LIN {X 0,Y 600.05,Z 1006.774,A -85,B 0,C 180,E1 28192.716,E2 28192.716} C_VEL
LIN {X 0,Y 598.178,Z 1023.897,A -85,B 0,C 180,E1 28190.857,E2 28190.857} C_VEL
LIN {X 0,Y 596.63,Z 1038.34,A -85,B 0,C 180,E1 28189.054,E2 28189.054} C_VEL
LIN {X 0,Y 595.296,Z 1052.251,A -85,B 0,C 180,E1 28187.094,E2 28187.094} C_VEL
LIN {X 0,Y 594.084,Z 1066.083,A -85,B 0,C 180,E1 28184.823,E2 28184.823} C_VEL
LIN {X 0,Y 593.249,Z 1077.838,A -85,B 0,C 180,E1 28182.61,E2 28182.61} C_VEL
LIN {X 0,Y 592.685,Z 1087.23,A -85,B 0,C 180,E1 28180.498,E2 28180.498} C_VEL
LIN {X 0,Y 592.308,Z 1095.363,A -85,B 0,C 180,E1 28178.348,E2 28178.348} C_VEL
LIN {X 0,Y 592.058,Z 1102.422,A -85,B 0,C 180,E1 28176.01,E2 28176.01} C_VEL
LIN {X 0,Y 591.967,Z 1107.243,A -85,B 0,C 180,E1 28173.971,E2 28173.971} C_VEL
LIN {X 0,Y 591.915,Z 1111.392,A -85,B 0,C 180,E1 28171.549,E2 28171.549} C_VEL
LIN {X 0,Y 591.912,Z 1113.53,A -85,B 0,C 180,E1 28169.419,E2 28169.419} C_VEL
LIN {X 0,Y 591.896,Z 1114.429,A -85,B 0,C 180,E1 28167.289,E2 28167.289} C_VEL
LIN {X 0,Y 591.895,Z 1113.793,A -85,B 0,C 180,E1 28164.863,E2 28164.863} C_VEL
LIN {X 0,Y 591.889,Z 1112.043,A -85,B 0,C 180,E1 28162.916,E2 28162.916} C_VEL
LIN {X 0,Y 591.93,Z 1109.042,A -85,B 0,C 180,E1 28160.864,E2 28160.864} C_VEL
LIN {X 0,Y 592.028,Z 1103.73,A -85,B 0,C 180,E1 28158.402,E2 28158.402} C_VEL
LIN {X 0,Y 592.196,Z 1098.141,A -85,B 0,C 180,E1 28156.426,E2 28156.426} C_VEL
LIN {X 0,Y 592.531,Z 1090.169,A -85,B 0,C 180,E1 28154.128,E2 28154.128} C_VEL
LIN {X 0,Y 593.026,Z 1080.989,A -85,B 0,C 180,E1 28151.981,E2 28151.981} C_VEL
LIN {X 0,Y 593.774,Z 1070.166,A -85,B 0,C 180,E1 28149.805,E2 28149.805} C_VEL
LIN {X 0,Y 594.831,Z 1057.029,A -85,B 0,C 180,E1 28147.568,E2 28147.568} C_VEL
LIN {X 0,Y 596.239,Z 1042.636,A -85,B 0,C 180,E1 28145.424,E2 28145.424} C_VEL
LIN {X 0,Y 597.762,Z 1027.606,A -85,B 0,C 180,E1 28143.497,E2 28143.497} C_VEL
LIN {X 0,Y 599.626,Z 1011.06,A -85,B 0,C 180,E1 28141.625,E2 28141.625} C_VEL
LIN {X 0,Y 601.534,Z 993.698,A -85,B 0,C 180,E1 28139.927,E2 28139.927} C_VEL
LIN {X 0,Y 603.744,Z 974.807,A -85,B 0,C 180,E1 28138.298,E2 28138.298} C_VEL
LIN {X 0,Y 605.898,Z 955.015,A -85,B 0,C 180,E1 28136.834,E2 28136.834} C_VEL
LIN {X 0,Y 608.034,Z 935.172,A -85,B 0,C 180,E1 28135.549,E2 28135.549} C_VEL
LIN {X 0,Y 610.125,Z 913.844,A -85,B 0,C 180,E1 28134.377,E2 28134.377} C_VEL
LIN {X 0,Y 611.917,Z 894.087,A -85,B 0,C 180,E1 28133.444,E2 28133.444} C_VEL
LIN {X 0,Y 613.892,Z 869.658,A -85,B 0,C 180,E1 28132.487,E2 28132.487} C_VEL
LIN {X 0,Y 615.266,Z 849.158,A -85,B 0,C 180,E1 28131.836,E2 28131.836} C_VEL
LIN {X 0,Y 616.599,Z 825.684,A -85,B 0,C 180,E1 28131.244,E2 28131.244} C_VEL
LIN {X 0,Y 617.493,Z 801.735,A -85,B 0,C 180,E1 28130.817,E2 28130.817} C_VEL
LIN {X 0,Y 622.364,Z 560.753,A -85,B 0,C 180,E1 28127.651,E2 28127.651} C_VEL
LIN {X 0,Y 624.229,Z 467.095,A -85,B 0,C 180,E1 28126.398,E2 28126.398} C_VEL
LIN {X 0,Y 610.775,Z 444.903,A -85,B 0,C 180,E1 28124.91,E2 28124.91} C_VEL
LIN {X 0,Y 602.614,Z 432.977,A -85,B 0,C 180,E1 28123.98,E2 28123.98} C_VEL
LIN {X 0,Y 599.127,Z 428.129,A -85,B 0,C 180,E1 28123.572,E2 28123.572} C_VEL
LIN {X 0,Y 596.004,Z 423.491,A -85,B 0,C 180,E1 28123.195,E2 28123.195} C_VEL
LIN {X 0,Y 593.804,Z 420.57,A -85,B 0,C 180,E1 28122.932,E2 28122.932} C_VEL
LIN {X 0,Y 593.243,Z 418.839,A -85,B 0,C 180,E1 28122.785,E2 28122.785} C_VEL
LIN {X 0,Y 593.129,Z 418.323,A -85,B 0,C 180,E1 28122.532,E2 28122.532} C_VEL
LIN {X 0,Y 593.115,Z 418.332,A -85,B 0,C 180,E1 28119.712,E2 28119.712} C_VEL
LIN {X 0,Y 593.141,Z 418.28,A -85,B 0,C 180,E1 28116.518,E2 28116.518} C_VEL
LIN {X 0,Y 593.127,Z 418.344,A -85,B 0,C 180,E1 28113.569,E2 28113.569} C_VEL
LIN {X 0,Y 593.136,Z 418.28,A -85,B 0,C 180,E1 28110.268,E2 28110.268} C_VEL
LIN {X 0,Y 593.14,Z 418.328,A -85,B 0,C 180,E1 28107.401,E2 28107.401} C_VEL
LIN {X 0,Y 593.144,Z 418.327,A -85,B 0,C 180,E1 28104.076,E2 28104.076} C_VEL
LIN {X 0,Y 593.163,Z 418.336,A -85,B 0,C 180,E1 28101.146,E2 28101.146} C_VEL
LIN {X 0,Y 593.149,Z 418.343,A -85,B 0,C 180,E1 28097.867,E2 28097.867} C_VEL
LIN {X 0,Y 593.202,Z 418.328,A -85,B 0,C 180,E1 28094.745,E2 28094.745} C_VEL
LIN {X 0,Y 593.148,Z 418.326,A -85,B 0,C 180,E1 28091.572,E2 28091.572} C_VEL
LIN {X 0,Y 593.199,Z 418.334,A -85,B 0,C 180,E1 28088.433,E2 28088.433} C_VEL
LIN {X 0,Y 593.159,Z 418.335,A -85,B 0,C 180,E1 28085.32,E2 28085.32} C_VEL
LIN {X 0,Y 593.189,Z 418.315,A -85,B 0,C 180,E1 28082.029,E2 28082.029} C_VEL
LIN {X 0,Y 593.193,Z 418.332,A -85,B 0,C 180,E1 28078.744,E2 28078.744} C_VEL
LIN {X 0,Y 593.172,Z 418.334,A -85,B 0,C 180,E1 28075.456,E2 28075.456} C_VEL
LIN {X 0,Y 593.189,Z 418.32,A -85,B 0,C 180,E1 28072.25,E2 28072.25} C_VEL
LIN {X 0,Y 593.178,Z 418.335,A -85,B 0,C 180,E1 28069.019,E2 28069.019} C_VEL
LIN {X 0,Y 593.199,Z 418.336,A -85,B 0,C 180,E1 28065.747,E2 28065.747} C_VEL
LIN {X 0,Y 593.19,Z 418.327,A -85,B 0,C 180,E1 28062.439,E2 28062.439} C_VEL
LIN {X 0,Y 593.183,Z 418.32,A -85,B 0,C 180,E1 28059.165,E2 28059.165} C_VEL
LIN {X 0,Y 593.18,Z 418.342,A -85,B 0,C 180,E1 28056.011,E2 28056.011} C_VEL
LIN {X 0,Y 593.188,Z 418.313,A -85,B 0,C 180,E1 28052.819,E2 28052.819} C_VEL
LIN {X 0,Y 593.177,Z 418.329,A -85,B 0,C 180,E1 28049.622,E2 28049.622} C_VEL
LIN {X 0,Y 593.187,Z 418.342,A -85,B 0,C 180,E1 28046.319,E2 28046.319} C_VEL
LIN {X 0,Y 593.197,Z 418.338,A -85,B 0,C 180,E1 28043.033,E2 28043.033} C_VEL
LIN {X 0,Y 593.161,Z 418.331,A -85,B 0,C 180,E1 28039.914,E2 28039.914} C_VEL
LIN {X 0,Y 593.211,Z 418.506,A -85,B 0,C 180,E1 28037.12,E2 28037.12} C_VEL
LIN {X 0,Y 597.822,Z 429.519,A -85,B 0,C 180,E1 28035.508,E2 28035.508} C_VEL
LIN {X 0,Y 605.197,Z 447.603,A -85,B 0,C 180,E1 28033.091,E2 28033.091} C_VEL
LIN {X 0,Y 606.689,Z 450.565,A -85,B 0,C 180,E1 28032.827,E2 28032.827} C_VEL
LIN {X 0,Y 617.614,Z 468.823,A -85,B 0,C 180,E1 28031.586,E2 28031.586} C_VEL
LIN {X 0,Y 620.789,Z 474.786,A -85,B 0,C 180,E1 28031.228,E2 28031.228} C_VEL
LIN {X 0,Y 624.171,Z 491.358,A -85,B 0,C 180,E1 28030.702,E2 28030.702} C_VEL
LIN {X 0,Y 619.361,Z 729.252,A -85,B 0,C 180,E1 28027.569,E2 28027.569} C_VEL
LIN {X 0,Y 617.111,Z 841.64,A -85,B 0,C 180,E1 28026.088,E2 28026.088} C_VEL
LIN {X 0,Y 615.922,Z 867.301,A -85,B 0,C 180,E1 28025.592,E2 28025.592} C_VEL
LIN {X 0,Y 614.631,Z 888.381,A -85,B 0,C 180,E1 28025.045,E2 28025.045} C_VEL
LIN {X 0,Y 612.923,Z 912.524,A -85,B 0,C 180,E1 28024.251,E2 28024.251} C_VEL
LIN {X 0,Y 611.154,Z 933.412,A -85,B 0,C 180,E1 28023.404,E2 28023.404} C_VEL
LIN {X 0,Y 609.26,Z 954.504,A -85,B 0,C 180,E1 28022.401,E2 28022.401} C_VEL
LIN {X 0,Y 607.047,Z 976.733,A -85,B 0,C 180,E1 28021.145,E2 28021.145} C_VEL
LIN {X 0,Y 605.079,Z 996.004,A -85,B 0,C 180,E1 28019.888,E2 28019.888} C_VEL
LIN {X 0,Y 602.838,Z 1016.85,A -85,B 0,C 180,E1 28018.319,E2 28018.319} C_VEL
LIN {X 0,Y 601,Z 1033.899,A -85,B 0,C 180,E1 28016.853,E2 28016.853} C_VEL
LIN {X 0,Y 598.954,Z 1053.455,A -85,B 0,C 180,E1 28014.931,E2 28014.931} C_VEL
LIN {X 0,Y 597.428,Z 1068.492,A -85,B 0,C 180,E1 28013.242,E2 28013.242} C_VEL
LIN {X 0,Y 595.881,Z 1084.893,A -85,B 0,C 180,E1 28011.148,E2 28011.148} C_VEL
LIN {X 0,Y 594.747,Z 1097.865,A -85,B 0,C 180,E1 28009.239,E2 28009.239} C_VEL
LIN {X 0,Y 593.777,Z 1110.217,A -85,B 0,C 180,E1 28007.139,E2 28007.139} C_VEL
LIN {X 0,Y 593.037,Z 1121.053,A -85,B 0,C 180,E1 28004.959,E2 28004.959} C_VEL
LIN {X 0,Y 592.515,Z 1130.773,A -85,B 0,C 180,E1 28002.673,E2 28002.673} C_VEL
LIN {X 0,Y 592.187,Z 1138.512,A -85,B 0,C 180,E1 28000.409,E2 28000.409} C_VEL
LIN {X 0,Y 592.024,Z 1144.591,A -85,B 0,C 180,E1 27998.222,E2 27998.222} C_VEL
LIN {X 0,Y 591.937,Z 1149.494,A -85,B 0,C 180,E1 27995.817,E2 27995.817} C_VEL
LIN {X 0,Y 591.915,Z 1152.349,A -85,B 0,C 180,E1 27993.777,E2 27993.777} C_VEL
LIN {X 0,Y 591.903,Z 1154.19,A -85,B 0,C 180,E1 27991.355,E2 27991.355} C_VEL
LIN {X 0,Y 591.885,Z 1154.349,A -85,B 0,C 180,E1 27989.322,E2 27989.322} C_VEL
LIN {X 0,Y 591.888,Z 1153.358,A -85,B 0,C 180,E1 27987.289,E2 27987.289} C_VEL
LIN {X 0,Y 591.902,Z 1150.611,A -85,B 0,C 180,E1 27984.863,E2 27984.863} C_VEL
LIN {X 0,Y 591.969,Z 1146.895,A -85,B 0,C 180,E1 27982.82,E2 27982.82} C_VEL
LIN {X 0,Y 592.092,Z 1141.711,A -85,B 0,C 180,E1 27980.67,E2 27980.67} C_VEL
LIN {X 0,Y 592.34,Z 1134.306,A -85,B 0,C 180,E1 27978.313,E2 27978.313} C_VEL
LIN {X 0,Y 592.697,Z 1126.746,A -85,B 0,C 180,E1 27976.339,E2 27976.339} C_VEL
LIN {X 0,Y 593.332,Z 1116.399,A -85,B 0,C 180,E1 27974.056,E2 27974.056} C_VEL
LIN {X 0,Y 594.113,Z 1105.682,A -85,B 0,C 180,E1 27972.062,E2 27972.062} C_VEL
LIN {X 0,Y 595.076,Z 1093.997,A -85,B 0,C 180,E1 27970.159,E2 27970.159} C_VEL
LIN {X 0,Y 596.424,Z 1078.851,A -85,B 0,C 180,E1 27968.046,E2 27968.046} C_VEL
LIN {X 0,Y 597.795,Z 1064.893,A -85,B 0,C 180,E1 27966.332,E2 27966.332} C_VEL
LIN {X 0,Y 599.722,Z 1046.098,A -85,B 0,C 180,E1 27964.311,E2 27964.311} C_VEL
LIN {X 0,Y 601.503,Z 1029.441,A -85,B 0,C 180,E1 27962.744,E2 27962.744} C_VEL
LIN {X 0,Y 603.743,Z 1008.537,A -85,B 0,C 180,E1 27961.025,E2 27961.025} C_VEL
LIN {X 0,Y 605.691,Z 989.997,A -85,B 0,C 180,E1 27959.699,E2 27959.699} C_VEL
LIN {X 0,Y 608.024,Z 967.457,A -85,B 0,C 180,E1 27958.304,E2 27958.304} C_VEL
LIN {X 0,Y 609.822,Z 948.512,A -85,B 0,C 180,E1 27957.298,E2 27957.298} C_VEL
LIN {X 0,Y 611.747,Z 927.152,A -85,B 0,C 180,E1 27956.32,E2 27956.32} C_VEL
LIN {X 0,Y 613.509,Z 903.939,A -85,B 0,C 180,E1 27955.447,E2 27955.447} C_VEL
LIN {X 0,Y 614.991,Z 882.112,A -85,B 0,C 180,E1 27954.779,E2 27954.779} C_VEL
LIN {X 0,Y 616.42,Z 856.718,A -85,B 0,C 180,E1 27954.191,E2 27954.191} C_VEL
LIN {X 0,Y 617.238,Z 834.898,A -85,B 0,C 180,E1 27953.824,E2 27953.824} C_VEL
LIN {X 0,Y 621.554,Z 599.011,A -85,B 0,C 180,E1 27950.762,E2 27950.762} C_VEL
LIN {X 0,Y 623.531,Z 489.86,A -85,B 0,C 180,E1 27949.324,E2 27949.324} C_VEL
LIN {X 0,Y 619.644,Z 473.187,A -85,B 0,C 180,E1 27948.779,E2 27948.779} C_VEL
LIN {X 0,Y 605.414,Z 448.968,A -85,B 0,C 180,E1 27947.25,E2 27947.25} C_VEL
LIN {X 0,Y 597.591,Z 429.213,A -85,B 0,C 180,E1 27944.783,E2 27944.783} C_VEL
LIN {X 0,Y 593.228,Z 418.535,A -85,B 0,C 180,E1 27943.318,E2 27943.318} C_VEL
LIN {X 0,Y 593.154,Z 418.284,A -85,B 0,C 180,E1 27940.34,E2 27940.34} C_VEL
LIN {X 0,Y 593.193,Z 418.324,A -85,B 0,C 180,E1 27937.239,E2 27937.239} C_VEL
LIN {X 0,Y 593.167,Z 418.338,A -85,B 0,C 180,E1 27934.031,E2 27934.031} C_VEL
LIN {X 0,Y 593.202,Z 418.338,A -85,B 0,C 180,E1 27930.723,E2 27930.723} C_VEL
LIN {X 0,Y 593.195,Z 418.331,A -85,B 0,C 180,E1 27927.398,E2 27927.398} C_VEL
LIN {X 0,Y 593.177,Z 418.316,A -85,B 0,C 180,E1 27924.181,E2 27924.181} C_VEL
LIN {X 0,Y 593.185,Z 418.337,A -85,B 0,C 180,E1 27921.041,E2 27921.041} C_VEL
LIN {X 0,Y 593.183,Z 418.33,A -85,B 0,C 180,E1 27917.764,E2 27917.764} C_VEL
LIN {X 0,Y 593.184,Z 418.318,A -85,B 0,C 180,E1 27914.546,E2 27914.546} C_VEL
LIN {X 0,Y 593.187,Z 418.341,A -85,B 0,C 180,E1 27911.175,E2 27911.175} C_VEL
LIN {X 0,Y 593.191,Z 418.317,A -85,B 0,C 180,E1 27907.945,E2 27907.945} C_VEL
LIN {X 0,Y 593.169,Z 418.332,A -85,B 0,C 180,E1 27904.738,E2 27904.738} C_VEL
LIN {X 0,Y 593.193,Z 418.329,A -85,B 0,C 180,E1 27901.545,E2 27901.545} C_VEL
LIN {X 0,Y 593.167,Z 418.325,A -85,B 0,C 180,E1 27898.409,E2 27898.409} C_VEL
LIN {X 0,Y 593.182,Z 418.343,A -85,B 0,C 180,E1 27895.068,E2 27895.068} C_VEL
LIN {X 0,Y 593.189,Z 418.313,A -85,B 0,C 180,E1 27891.86,E2 27891.86} C_VEL
LIN {X 0,Y 593.155,Z 418.34,A -85,B 0,C 180,E1 27888.625,E2 27888.625} C_VEL
LIN {X 0,Y 593.2,Z 418.317,A -85,B 0,C 180,E1 27885.454,E2 27885.454} C_VEL
LIN {X 0,Y 593.144,Z 418.334,A -85,B 0,C 180,E1 27882.336,E2 27882.336} C_VEL
LIN {X 0,Y 593.199,Z 418.335,A -85,B 0,C 180,E1 27879.166,E2 27879.166} C_VEL
LIN {X 0,Y 593.136,Z 418.318,A -85,B 0,C 180,E1 27876.135,E2 27876.135} C_VEL
LIN {X 0,Y 593.177,Z 418.335,A -85,B 0,C 180,E1 27872.927,E2 27872.927} C_VEL
LIN {X 0,Y 593.132,Z 418.342,A -85,B 0,C 180,E1 27869.955,E2 27869.955} C_VEL
LIN {X 0,Y 593.156,Z 418.328,A -85,B 0,C 180,E1 27866.732,E2 27866.732} C_VEL
LIN {X 0,Y 593.125,Z 418.338,A -85,B 0,C 180,E1 27863.841,E2 27863.841} C_VEL
LIN {X 0,Y 593.152,Z 418.339,A -85,B 0,C 180,E1 27860.666,E2 27860.666} C_VEL
LIN {X 0,Y 593.104,Z 418.276,A -85,B 0,C 180,E1 27857.858,E2 27857.858} C_VEL
LIN {X 0,Y 593.152,Z 418.346,A -85,B 0,C 180,E1 27854.653,E2 27854.653} C_VEL
LIN {X 0,Y 593.097,Z 418.282,A -85,B 0,C 180,E1 27851.682,E2 27851.682} C_VEL
LIN {X 0,Y 593.209,Z 418.548,A -85,B 0,C 180,E1 27850.844,E2 27850.844} C_VEL
LIN {X 0,Y 593.536,Z 419.937,A -85,B 0,C 180,E1 27850.687,E2 27850.687} C_VEL
LIN {X 0,Y 595.547,Z 423.115,A -85,B 0,C 180,E1 27850.449,E2 27850.449} C_VEL
LIN {X 0,Y 596.796,Z 424.91,A -85,B 0,C 180,E1 27850.31,E2 27850.31} C_VEL
LIN {X 0,Y 607.889,Z 441.301,A -85,B 0,C 180,E1 27849.107,E2 27849.107} C_VEL
LIN {X 0,Y 623.849,Z 467.241,A -85,B 0,C 180,E1 27847.442,E2 27847.442} C_VEL
LIN {X 0,Y 622.311,Z 544.948,A -85,B 0,C 180,E1 27846.423,E2 27846.423} C_VEL
LIN {X 0,Y 621.357,Z 552.646,A -85,B 0,C 180,E1 27846.382,E2 27846.382} C_VEL
LIN {X 0,Y 616.074,Z 573.201,A -85,B 0,C 180,E1 27846.476,E2 27846.476} C_VEL
LIN {X 0,Y 615.373,Z 579.803,A -85,B 0,C 180,E1 27846.432,E2 27846.432} C_VEL
LIN {X 0,Y 610.821,Z 804.731,A -85,B 0,C 180,E1 27843.476,E2 27843.476} C_VEL
LIN {X 0,Y 609.717,Z 830.998,A -85,B 0,C 180,E1 27842.97,E2 27842.97} C_VEL
LIN {X 0,Y 608.493,Z 851.442,A -85,B 0,C 180,E1 27842.436,E2 27842.436} C_VEL
LIN {X 0,Y 606.891,Z 874.614,A -85,B 0,C 180,E1 27841.679,E2 27841.679} C_VEL
LIN {X 0,Y 604.931,Z 896.78,A -85,B 0,C 180,E1 27840.774,E2 27840.774} C_VEL
LIN {X 0,Y 602.985,Z 917.369,A -85,B 0,C 180,E1 27839.778,E2 27839.778} C_VEL
LIN {X 0,Y 600.686,Z 938.996,A -85,B 0,C 180,E1 27838.538,E2 27838.538} C_VEL
LIN {X 0,Y 598.657,Z 957.009,A -85,B 0,C 180,E1 27837.343,E2 27837.343} C_VEL
LIN {X 0,Y 596.2,Z 977.938,A -85,B 0,C 180,E1 27835.745,E2 27835.745} C_VEL
LIN {X 0,Y 594.122,Z 994.981,A -85,B 0,C 180,E1 27834.245,E2 27834.245} C_VEL
LIN {X 0,Y 592.002,Z 1013.013,A -85,B 0,C 180,E1 27832.44,E2 27832.44} C_VEL
LIN {X 0,Y 590.145,Z 1028.649,A -85,B 0,C 180,E1 27830.635,E2 27830.635} C_VEL
LIN {X 0,Y 588.491,Z 1043.984,A -85,B 0,C 180,E1 27828.628,E2 27828.628} C_VEL
LIN {X 0,Y 587.102,Z 1057.157,A -85,B 0,C 180,E1 27826.626,E2 27826.626} C_VEL
LIN {X 0,Y 586.026,Z 1069.289,A -85,B 0,C 180,E1 27824.526,E2 27824.526} C_VEL
LIN {X 0,Y 585.142,Z 1080.722,A -85,B 0,C 180,E1 27822.194,E2 27822.194} C_VEL
LIN {X 0,Y 584.612,Z 1089.812,A -85,B 0,C 180,E1 27820.047,E2 27820.047} C_VEL
LIN {X 0,Y 584.237,Z 1098.008,A -85,B 0,C 180,E1 27817.672,E2 27817.672} C_VEL
LIN {X 0,Y 584.035,Z 1103.796,A -85,B 0,C 180,E1 27815.6,E2 27815.6} C_VEL
LIN {X 0,Y 583.929,Z 1109.024,A -85,B 0,C 180,E1 27813.141,E2 27813.141} C_VEL
LIN {X 0,Y 583.893,Z 1112.005,A -85,B 0,C 180,E1 27811.079,E2 27811.079} C_VEL
LIN {X 0,Y 583.9,Z 1113.762,A -85,B 0,C 180,E1 27809.117,E2 27809.117} C_VEL
LIN {X 0,Y 583.895,Z 1114.44,A -85,B 0,C 180,E1 27806.662,E2 27806.662} C_VEL
LIN {X 0,Y 583.908,Z 1113.559,A -85,B 0,C 180,E1 27804.497,E2 27804.497} C_VEL
LIN {X 0,Y 583.925,Z 1111.424,A -85,B 0,C 180,E1 27802.324,E2 27802.324} C_VEL
LIN {X 0,Y 583.977,Z 1107.242,A -85,B 0,C 180,E1 27799.842,E2 27799.842} C_VEL
LIN {X 0,Y 584.067,Z 1102.564,A -85,B 0,C 180,E1 27797.83,E2 27797.83} C_VEL
LIN {X 0,Y 584.339,Z 1095.46,A -85,B 0,C 180,E1 27795.431,E2 27795.431} C_VEL
LIN {X 0,Y 584.754,Z 1087.143,A -85,B 0,C 180,E1 27793.203,E2 27793.203} C_VEL
LIN {X 0,Y 585.402,Z 1077.256,A -85,B 0,C 180,E1 27790.959,E2 27790.959} C_VEL
LIN {X 0,Y 586.294,Z 1066.066,A -85,B 0,C 180,E1 27788.804,E2 27788.804} C_VEL
LIN {X 0,Y 587.469,Z 1053.823,A -85,B 0,C 180,E1 27786.742,E2 27786.742} C_VEL
LIN {X 0,Y 588.944,Z 1039.5,A -85,B 0,C 180,E1 27784.669,E2 27784.669} C_VEL
LIN {X 0,Y 590.513,Z 1025.638,A -85,B 0,C 180,E1 27782.904,E2 27782.904} C_VEL
LIN {X 0,Y 592.594,Z 1007.842,A -85,B 0,C 180,E1 27780.925,E2 27780.925} C_VEL
LIN {X 0,Y 594.618,Z 991.223,A -85,B 0,C 180,E1 27779.312,E2 27779.312} C_VEL
LIN {X 0,Y 597.05,Z 970.874,A -85,B 0,C 180,E1 27777.594,E2 27777.594} C_VEL
LIN {X 0,Y 599.106,Z 953.171,A -85,B 0,C 180,E1 27776.294,E2 27776.294} C_VEL
LIN {X 0,Y 601.587,Z 931.163,A -85,B 0,C 180,E1 27774.894,E2 27774.894} C_VEL
LIN {X 0,Y 603.541,Z 912.109,A -85,B 0,C 180,E1 27773.858,E2 27773.858} C_VEL
LIN {X 0,Y 605.588,Z 890.917,A -85,B 0,C 180,E1 27772.864,E2 27772.864} C_VEL
LIN {X 0,Y 607.464,Z 867.705,A -85,B 0,C 180,E1 27771.974,E2 27771.974} C_VEL
LIN {X 0,Y 608.969,Z 846.238,A -85,B 0,C 180,E1 27771.301,E2 27771.301} C_VEL
LIN {X 0,Y 610.364,Z 821.032,A -85,B 0,C 180,E1 27770.701,E2 27770.701} C_VEL
LIN {X 0,Y 611.203,Z 799.034,A -85,B 0,C 180,E1 27770.323,E2 27770.323} C_VEL
LIN {X 0,Y 616.602,Z 546.316,A -85,B 0,C 180,E1 27766.975,E2 27766.975} C_VEL
LIN {X 0,Y 618.221,Z 470.366,A -85,B 0,C 180,E1 27765.949,E2 27765.949} C_VEL
LIN {X 0,Y 605.233,Z 449.14,A -85,B 0,C 180,E1 27764.482,E2 27764.482} C_VEL
LIN {X 0,Y 597.704,Z 438.133,A -85,B 0,C 180,E1 27763.603,E2 27763.603} C_VEL
LIN {X 0,Y 591.444,Z 429.254,A -85,B 0,C 180,E1 27762.847,E2 27762.847} C_VEL
LIN {X 0,Y 588.36,Z 424.737,A -85,B 0,C 180,E1 27762.463,E2 27762.463} C_VEL
LIN {X 0,Y 585.933,Z 421.842,A -85,B 0,C 180,E1 27762.167,E2 27762.167} C_VEL
LIN {X 0,Y 585.242,Z 419.789,A -85,B 0,C 180,E1 27761.995,E2 27761.995} C_VEL
LIN {X 0,Y 585.172,Z 419.275,A -85,B 0,C 180,E1 27761.659,E2 27761.659} C_VEL
LIN {X 0,Y 585.186,Z 419.32,A -85,B 0,C 180,E1 27758.334,E2 27758.334} C_VEL
LIN {X 0,Y 585.194,Z 419.272,A -85,B 0,C 180,E1 27755.397,E2 27755.397} C_VEL
LIN {X 0,Y 585.19,Z 419.323,A -85,B 0,C 180,E1 27752.1,E2 27752.1} C_VEL
LIN {X 0,Y 585.22,Z 419.262,A -85,B 0,C 180,E1 27749.14,E2 27749.14} C_VEL
LIN {X 0,Y 585.197,Z 419.335,A -85,B 0,C 180,E1 27745.939,E2 27745.939} C_VEL
LIN {X 0,Y 585.26,Z 419.323,A -85,B 0,C 180,E1 27742.819,E2 27742.819} C_VEL
LIN {X 0,Y 585.201,Z 419.317,A -85,B 0,C 180,E1 27739.67,E2 27739.67} C_VEL
LIN {X 0,Y 585.258,Z 419.308,A -85,B 0,C 180,E1 27736.476,E2 27736.476} C_VEL
LIN {X 0,Y 585.215,Z 419.334,A -85,B 0,C 180,E1 27733.336,E2 27733.336} C_VEL
LIN {X 0,Y 585.237,Z 419.327,A -85,B 0,C 180,E1 27730.036,E2 27730.036} C_VEL
LIN {X 0,Y 585.247,Z 419.31,A -85,B 0,C 180,E1 27726.869,E2 27726.869} C_VEL
LIN {X 0,Y 585.225,Z 419.328,A -85,B 0,C 180,E1 27723.624,E2 27723.624} C_VEL
LIN {X 0,Y 585.257,Z 419.323,A -85,B 0,C 180,E1 27720.392,E2 27720.392} C_VEL
LIN {X 0,Y 585.227,Z 419.307,A -85,B 0,C 180,E1 27717.16,E2 27717.16} C_VEL
LIN {X 0,Y 585.255,Z 419.317,A -85,B 0,C 180,E1 27713.821,E2 27713.821} C_VEL
LIN {X 0,Y 585.254,Z 419.33,A -85,B 0,C 180,E1 27710.461,E2 27710.461} C_VEL
LIN {X 0,Y 585.236,Z 419.31,A -85,B 0,C 180,E1 27707.167,E2 27707.167} C_VEL
LIN {X 0,Y 585.245,Z 419.314,A -85,B 0,C 180,E1 27704.034,E2 27704.034} C_VEL
LIN {X 0,Y 585.252,Z 419.332,A -85,B 0,C 180,E1 27700.747,E2 27700.747} C_VEL
LIN {X 0,Y 585.258,Z 419.306,A -85,B 0,C 180,E1 27697.393,E2 27697.393} C_VEL
LIN {X 0,Y 585.239,Z 419.309,A -85,B 0,C 180,E1 27694.172,E2 27694.172} C_VEL
LIN {X 0,Y 585.252,Z 419.329,A -85,B 0,C 180,E1 27690.974,E2 27690.974} C_VEL
LIN {X 0,Y 585.23,Z 419.314,A -85,B 0,C 180,E1 27687.787,E2 27687.787} C_VEL
LIN {X 0,Y 585.255,Z 419.306,A -85,B 0,C 180,E1 27684.582,E2 27684.582} C_VEL
LIN {X 0,Y 585.241,Z 419.311,A -85,B 0,C 180,E1 27681.333,E2 27681.333} C_VEL
LIN {X 0,Y 585.23,Z 419.357,A -85,B 0,C 180,E1 27678.006,E2 27678.006} C_VEL
LIN {X 0,Y 585.303,Z 419.848,A -85,B 0,C 180,E1 27677.785,E2 27677.785} C_VEL
LIN {X 0,Y 592.102,Z 435.669,A -85,B 0,C 180,E1 27675.45,E2 27675.45} C_VEL
LIN {X 0,Y 597.515,Z 448.594,A -85,B 0,C 180,E1 27673.719,E2 27673.719} C_VEL
LIN {X 0,Y 610.489,Z 470.096,A -85,B 0,C 180,E1 27672.179,E2 27672.179} C_VEL
LIN {X 0,Y 615.277,Z 478.799,A -85,B 0,C 180,E1 27671.63,E2 27671.63} C_VEL
LIN {X 0,Y 618.124,Z 493.199,A -85,B 0,C 180,E1 27671.168,E2 27671.168} C_VEL
LIN {X 0,Y 613.047,Z 730.309,A -85,B 0,C 180,E1 27668.017,E2 27668.017} C_VEL
LIN {X 0,Y 610.688,Z 841.32,A -85,B 0,C 180,E1 27666.539,E2 27666.539} C_VEL
LIN {X 0,Y 609.414,Z 867.194,A -85,B 0,C 180,E1 27666.036,E2 27666.036} C_VEL
LIN {X 0,Y 608.038,Z 888.463,A -85,B 0,C 180,E1 27665.478,E2 27665.478} C_VEL
LIN {X 0,Y 606.24,Z 912.394,A -85,B 0,C 180,E1 27664.682,E2 27664.682} C_VEL
LIN {X 0,Y 604.378,Z 933.221,A -85,B 0,C 180,E1 27663.829,E2 27663.829} C_VEL
LIN {X 0,Y 602.37,Z 954.246,A -85,B 0,C 180,E1 27662.818,E2 27662.818} C_VEL
LIN {X 0,Y 600.014,Z 976.431,A -85,B 0,C 180,E1 27661.552,E2 27661.552} C_VEL
LIN {X 0,Y 597.92,Z 995.771,A -85,B 0,C 180,E1 27660.278,E2 27660.278} C_VEL
LIN {X 0,Y 595.564,Z 1016.545,A -85,B 0,C 180,E1 27658.696,E2 27658.696} C_VEL
LIN {X 0,Y 593.589,Z 1033.748,A -85,B 0,C 180,E1 27657.201,E2 27657.201} C_VEL
LIN {X 0,Y 591.377,Z 1053.62,A -85,B 0,C 180,E1 27655.219,E2 27655.219} C_VEL
LIN {X 0,Y 589.732,Z 1068.861,A -85,B 0,C 180,E1 27653.481,E2 27653.481} C_VEL
LIN {X 0,Y 588.039,Z 1085.699,A -85,B 0,C 180,E1 27651.281,E2 27651.281} C_VEL
LIN {X 0,Y 586.881,Z 1098.212,A -85,B 0,C 180,E1 27649.404,E2 27649.404} C_VEL
LIN {X 0,Y 585.79,Z 1111.701,A -85,B 0,C 180,E1 27647.073,E2 27647.073} C_VEL
LIN {X 0,Y 585.131,Z 1121.094,A -85,B 0,C 180,E1 27645.156,E2 27645.156} C_VEL
LIN {X 0,Y 584.57,Z 1130.783,A -85,B 0,C 180,E1 27642.845,E2 27642.845} C_VEL
LIN {X 0,Y 584.217,Z 1138.512,A -85,B 0,C 180,E1 27640.552,E2 27640.552} C_VEL
LIN {X 0,Y 584.036,Z 1144.718,A -85,B 0,C 180,E1 27638.286,E2 27638.286} C_VEL
LIN {X 0,Y 583.944,Z 1149.494,A -85,B 0,C 180,E1 27635.897,E2 27635.897} C_VEL
LIN {X 0,Y 583.915,Z 1152.349,A -85,B 0,C 180,E1 27633.829,E2 27633.829} C_VEL
LIN {X 0,Y 583.902,Z 1154.19,A -85,B 0,C 180,E1 27631.374,E2 27631.374} C_VEL
LIN {X 0,Y 583.885,Z 1154.348,A -85,B 0,C 180,E1 27629.313,E2 27629.313} C_VEL
LIN {X 0,Y 583.89,Z 1153.426,A -85,B 0,C 180,E1 27627.35,E2 27627.35} C_VEL
LIN {X 0,Y 583.905,Z 1150.929,A -85,B 0,C 180,E1 27624.99,E2 27624.99} C_VEL
LIN {X 0,Y 583.971,Z 1147.101,A -85,B 0,C 180,E1 27622.82,E2 27622.82} C_VEL
LIN {X 0,Y 584.086,Z 1142.219,A -85,B 0,C 180,E1 27620.74,E2 27620.74} C_VEL
LIN {X 0,Y 584.365,Z 1134.658,A -85,B 0,C 180,E1 27618.251,E2 27618.251} C_VEL
LIN {X 0,Y 584.746,Z 1127.072,A -85,B 0,C 180,E1 27616.23,E2 27616.23} C_VEL
LIN {X 0,Y 585.417,Z 1116.912,A -85,B 0,C 180,E1 27613.937,E2 27613.937} C_VEL
LIN {X 0,Y 586.225,Z 1106.102,A -85,B 0,C 180,E1 27611.915,E2 27611.915} C_VEL
LIN {X 0,Y 587.232,Z 1094.351,A -85,B 0,C 180,E1 27609.986,E2 27609.986} C_VEL
LIN {X 0,Y 588.656,Z 1079.34,A -85,B 0,C 180,E1 27607.846,E2 27607.846} C_VEL
LIN {X 0,Y 590.1,Z 1065.458,A -85,B 0,C 180,E1 27606.11,E2 27606.11} C_VEL
LIN {X 0,Y 592.031,Z 1047.857,A -85,B 0,C 180,E1 27604.167,E2 27604.167} C_VEL
LIN {X 0,Y 593.957,Z 1030.723,A -85,B 0,C 180,E1 27602.521,E2 27602.521} C_VEL
LIN {X 0,Y 596.169,Z 1011.618,A -85,B 0,C 180,E1 27600.897,E2 27600.897} C_VEL
LIN {X 0,Y 598.313,Z 992.123,A -85,B 0,C 180,E1 27599.467,E2 27599.467} C_VEL
LIN {X 0,Y 600.595,Z 971.593,A -85,B 0,C 180,E1 27598.146,E2 27598.146} C_VEL
LIN {X 0,Y 602.753,Z 950.216,A -85,B 0,C 180,E1 27596.979,E2 27596.979} C_VEL
LIN {X 0,Y 604.474,Z 931.982,A -85,B 0,C 180,E1 27596.12,E2 27596.12} C_VEL
LIN {X 0,Y 606.477,Z 908.711,A -85,B 0,C 180,E1 27595.19,E2 27595.19} C_VEL
LIN {X 0,Y 608.102,Z 885.734,A -85,B 0,C 180,E1 27594.457,E2 27594.457} C_VEL
LIN {X 0,Y 609.617,Z 861.627,A -85,B 0,C 180,E1 27593.853,E2 27593.853} C_VEL
LIN {X 0,Y 610.635,Z 837.267,A -85,B 0,C 180,E1 27593.424,E2 27593.424} C_VEL
LIN {X 0,Y 615.209,Z 602.161,A -85,B 0,C 180,E1 27590.342,E2 27590.342} C_VEL
LIN {X 0,Y 617.3,Z 491.496,A -85,B 0,C 180,E1 27588.868,E2 27588.868} C_VEL
LIN {X 0,Y 613.962,Z 477.24,A -85,B 0,C 180,E1 27588.394,E2 27588.394} C_VEL
LIN {X 0,Y 599.58,Z 452.97,A -85,B 0,C 180,E1 27586.835,E2 27586.835} C_VEL
LIN {X 0,Y 596.897,Z 448.207,A -85,B 0,C 180,E1 27586.489,E2 27586.489} C_VEL
LIN {X 0,Y 589.654,Z 430.249,A -85,B 0,C 180,E1 27584.168,E2 27584.168} C_VEL
LIN {X 0,Y 585.256,Z 419.491,A -85,B 0,C 180,E1 27582.651,E2 27582.651} C_VEL
LIN {X 0,Y 585.241,Z 419.287,A -85,B 0,C 180,E1 27579.716,E2 27579.716} C_VEL
LIN {X 0,Y 585.23,Z 419.312,A -85,B 0,C 180,E1 27576.416,E2 27576.416} C_VEL
LIN {X 0,Y 585.255,Z 419.31,A -85,B 0,C 180,E1 27573.259,E2 27573.259} C_VEL
LIN {X 0,Y 585.229,Z 419.327,A -85,B 0,C 180,E1 27570.04,E2 27570.04} C_VEL
LIN {X 0,Y 585.255,Z 419.328,A -85,B 0,C 180,E1 27566.81,E2 27566.81} C_VEL
LIN {X 0,Y 585.255,Z 419.306,A -85,B 0,C 180,E1 27563.443,E2 27563.443} C_VEL
LIN {X 0,Y 585.247,Z 419.32,A -85,B 0,C 180,E1 27560.189,E2 27560.189} C_VEL
LIN {X 0,Y 585.244,Z 419.33,A -85,B 0,C 180,E1 27556.909,E2 27556.909} C_VEL
LIN {X 0,Y 585.244,Z 419.304,A -85,B 0,C 180,E1 27553.738,E2 27553.738} C_VEL
LIN {X 0,Y 585.243,Z 419.323,A -85,B 0,C 180,E1 27550.534,E2 27550.534} C_VEL
LIN {X 0,Y 585.249,Z 419.319,A -85,B 0,C 180,E1 27547.165,E2 27547.165} C_VEL
LIN {X 0,Y 585.253,Z 419.31,A -85,B 0,C 180,E1 27543.919,E2 27543.919} C_VEL
LIN {X 0,Y 585.227,Z 419.331,A -85,B 0,C 180,E1 27540.685,E2 27540.685} C_VEL
LIN {X 0,Y 585.253,Z 419.303,A -85,B 0,C 180,E1 27537.454,E2 27537.454} C_VEL
LIN {X 0,Y 585.229,Z 419.328,A -85,B 0,C 180,E1 27534.214,E2 27534.214} C_VEL
LIN {X 0,Y 585.227,Z 419.314,A -85,B 0,C 180,E1 27530.857,E2 27530.857} C_VEL
LIN {X 0,Y 585.256,Z 419.319,A -85,B 0,C 180,E1 27527.669,E2 27527.669} C_VEL
LIN {X 0,Y 585.21,Z 419.332,A -85,B 0,C 180,E1 27524.505,E2 27524.505} C_VEL
LIN {X 0,Y 585.259,Z 419.306,A -85,B 0,C 180,E1 27521.368,E2 27521.368} C_VEL
LIN {X 0,Y 585.2,Z 419.331,A -85,B 0,C 180,E1 27518.237,E2 27518.237} C_VEL
LIN {X 0,Y 585.247,Z 419.312,A -85,B 0,C 180,E1 27515.039,E2 27515.039} C_VEL
LIN {X 0,Y 585.196,Z 419.318,A -85,B 0,C 180,E1 27511.974,E2 27511.974} C_VEL
LIN {X 0,Y 585.214,Z 419.33,A -85,B 0,C 180,E1 27508.682,E2 27508.682} C_VEL
LIN {X 0,Y 585.201,Z 419.331,A -85,B 0,C 180,E1 27505.677,E2 27505.677} C_VEL
LIN {X 0,Y 585.19,Z 419.326,A -85,B 0,C 180,E1 27502.411,E2 27502.411} C_VEL
LIN {X 0,Y 585.184,Z 419.295,A -85,B 0,C 180,E1 27499.64,E2 27499.64} C_VEL
LIN {X 0,Y 585.173,Z 419.287,A -85,B 0,C 180,E1 27496.285,E2 27496.285} C_VEL
LIN {X 0,Y 585.186,Z 419.289,A -85,B 0,C 180,E1 27493.384,E2 27493.384} C_VEL
LIN {X 0,Y 585.189,Z 419.452,A -85,B 0,C 180,E1 27491.585,E2 27491.585} C_VEL
LIN {X 0,Y 585.536,Z 420.845,A -85,B 0,C 180,E1 27491.402,E2 27491.402} C_VEL
LIN {X 0,Y 587.43,Z 423.887,A -85,B 0,C 180,E1 27491.168,E2 27491.168} C_VEL
LIN {X 0,Y 588.76,Z 425.467,A -85,B 0,C 180,E1 27491.021,E2 27491.021} C_VEL
LIN {X 0,Y 591.543,Z 429.527,A -85,B 0,C 180,E1 27490.702,E2 27490.702} C_VEL
LIN {X 0,Y 605.321,Z 450.203,A -85,B 0,C 180,E1 27489.183,E2 27489.183} C_VEL
LIN {X 0,Y 617.641,Z 470.603,A -85,B 0,C 180,E1 27487.874,E2 27487.874} C_VEL
LIN {X 0,Y 615.373,Z 579.803,A -85,B 0,C 180,E1 27486.432,E2 27486.432} C_VEL
LIN {X 0,Y 614.451,Z 587.499,A -85,B 0,C 180,E1 27486.388,E2 27486.388} C_VEL
LIN {X 0,Y 609.124,Z 608.05,A -85,B 0,C 180,E1 27486.486,E2 27486.486} C_VEL
LIN {X 0,Y 608.406,Z 614.655,A -85,B 0,C 180,E1 27486.442,E2 27486.442} C_VEL
LIN {X 0,Y 604.328,Z 805.826,A -85,B 0,C 180,E1 27483.907,E2 27483.907} C_VEL
LIN {X 0,Y 603.172,Z 831.725,A -85,B 0,C 180,E1 27483.399,E2 27483.399} C_VEL
LIN {X 0,Y 601.898,Z 852.117,A -85,B 0,C 180,E1 27482.861,E2 27482.861} C_VEL
LIN {X 0,Y 600.227,Z 875.132,A -85,B 0,C 180,E1 27482.101,E2 27482.101} C_VEL
LIN {X 0,Y 598.234,Z 896.836,A -85,B 0,C 180,E1 27481.207,E2 27481.207} C_VEL
LIN {X 0,Y 596.306,Z 916.322,A -85,B 0,C 180,E1 27480.263,E2 27480.263} C_VEL
LIN {X 0,Y 593.783,Z 939.121,A -85,B 0,C 180,E1 27478.956,E2 27478.956} C_VEL
LIN {X 0,Y 591.567,Z 957.896,A -85,B 0,C 180,E1 27477.698,E2 27477.698} C_VEL
LIN {X 0,Y 588.906,Z 979.323,A -85,B 0,C 180,E1 27476.034,E2 27476.034} C_VEL
LIN {X 0,Y 586.799,Z 995.731,A -85,B 0,C 180,E1 27474.568,E2 27474.568} C_VEL
LIN {X 0,Y 584.554,Z 1013.69,A -85,B 0,C 180,E1 27472.742,E2 27472.742} C_VEL
LIN {X 0,Y 582.596,Z 1029.29,A -85,B 0,C 180,E1 27470.915,E2 27470.915} C_VEL
LIN {X 0,Y 580.831,Z 1044.568,A -85,B 0,C 180,E1 27468.883,E2 27468.883} C_VEL
LIN {X 0,Y 579.357,Z 1057.713,A -85,B 0,C 180,E1 27466.855,E2 27466.855} C_VEL
LIN {X 0,Y 578.211,Z 1069.817,A -85,B 0,C 180,E1 27464.727,E2 27464.727} C_VEL
LIN {X 0,Y 577.303,Z 1080.504,A -85,B 0,C 180,E1 27462.504,E2 27462.504} C_VEL
LIN {X 0,Y 576.718,Z 1089.234,A -85,B 0,C 180,E1 27460.388,E2 27460.388} C_VEL
LIN {X 0,Y 576.283,Z 1097.535,A -85,B 0,C 180,E1 27457.979,E2 27457.979} C_VEL
LIN {X 0,Y 576.056,Z 1103.398,A -85,B 0,C 180,E1 27455.878,E2 27455.878} C_VEL
LIN {X 0,Y 575.94,Z 1108.444,A -85,B 0,C 180,E1 27453.583,E2 27453.583} C_VEL
LIN {X 0,Y 575.9,Z 1111.827,A -85,B 0,C 180,E1 27451.293,E2 27451.293} C_VEL
LIN {X 0,Y 575.91,Z 1113.655,A -85,B 0,C 180,E1 27449.304,E2 27449.304} C_VEL
LIN {X 0,Y 575.904,Z 1114.497,A -85,B 0,C 180,E1 27446.915,E2 27446.915} C_VEL
LIN {X 0,Y 575.907,Z 1113.666,A -85,B 0,C 180,E1 27444.62,E2 27444.62} C_VEL
LIN {X 0,Y 575.899,Z 1111.831,A -85,B 0,C 180,E1 27442.618,E2 27442.618} C_VEL
LIN {X 0,Y 575.942,Z 1108.402,A -85,B 0,C 180,E1 27440.305,E2 27440.305} C_VEL
LIN {X 0,Y 576.049,Z 1103.519,A -85,B 0,C 180,E1 27438.079,E2 27438.079} C_VEL
LIN {X 0,Y 576.268,Z 1097.876,A -85,B 0,C 180,E1 27436.044,E2 27436.044} C_VEL
LIN {X 0,Y 576.701,Z 1089.478,A -85,B 0,C 180,E1 27433.584,E2 27433.584} C_VEL
LIN {X 0,Y 577.3,Z 1080.554,A -85,B 0,C 180,E1 27431.416,E2 27431.416} C_VEL
LIN {X 0,Y 578.239,Z 1069.547,A -85,B 0,C 180,E1 27429.132,E2 27429.132} C_VEL
LIN {X 0,Y 579.369,Z 1057.658,A -85,B 0,C 180,E1 27427.043,E2 27427.043} C_VEL
LIN {X 0,Y 580.903,Z 1044.07,A -85,B 0,C 180,E1 27424.948,E2 27424.948} C_VEL
LIN {X 0,Y 582.648,Z 1028.964,A -85,B 0,C 180,E1 27422.95,E2 27422.95} C_VEL
LIN {X 0,Y 584.611,Z 1013.384,A -85,B 0,C 180,E1 27421.129,E2 27421.129} C_VEL
LIN {X 0,Y 586.845,Z 995.508,A -85,B 0,C 180,E1 27419.316,E2 27419.316} C_VEL
LIN {X 0,Y 589.056,Z 978.397,A -85,B 0,C 180,E1 27417.792,E2 27417.792} C_VEL
LIN {X 0,Y 591.667,Z 957.309,A -85,B 0,C 180,E1 27416.162,E2 27416.162} C_VEL
LIN {X 0,Y 593.914,Z 938.555,A -85,B 0,C 180,E1 27414.906,E2 27414.906} C_VEL
LIN {X 0,Y 596.471,Z 915.739,A -85,B 0,C 180,E1 27413.599,E2 27413.599} C_VEL
LIN {X 0,Y 598.426,Z 896.448,A -85,B 0,C 180,E1 27412.661,E2 27412.661} C_VEL
LIN {X 0,Y 600.54,Z 873.751,A -85,B 0,C 180,E1 27411.729,E2 27411.729} C_VEL
LIN {X 0,Y 602.205,Z 851.292,A -85,B 0,C 180,E1 27410.99,E2 27410.99} C_VEL
LIN {X 0,Y 603.559,Z 830.091,A -85,B 0,C 180,E1 27410.432,E2 27410.432} C_VEL
LIN {X 0,Y 604.689,Z 804.624,A -85,B 0,C 180,E1 27409.943,E2 27409.943} C_VEL
LIN {X 0,Y 610.012,Z 570.914,A -85,B 0,C 180,E1 27406.81,E2 27406.81} C_VEL
LIN {X 0,Y 612.177,Z 473.5,A -85,B 0,C 180,E1 27405.483,E2 27405.483} C_VEL
LIN {X 0,Y 599.275,Z 452.543,A -85,B 0,C 180,E1 27403.989,E2 27403.989} C_VEL
LIN {X 0,Y 590.483,Z 439.918,A -85,B 0,C 180,E1 27402.934,E2 27402.934} C_VEL
LIN {X 0,Y 583.996,Z 430.758,A -85,B 0,C 180,E1 27402.124,E2 27402.124} C_VEL
LIN {X 0,Y 581.244,Z 426.926,A -85,B 0,C 180,E1 27401.773,E2 27401.773} C_VEL
LIN {X 0,Y 580.331,Z 425.644,A -85,B 0,C 180,E1 27401.655,E2 27401.655} C_VEL
LIN {X 0,Y 578.027,Z 422.821,A -85,B 0,C 180,E1 27401.361,E2 27401.361} C_VEL
LIN {X 0,Y 577.368,Z 420.81,A -85,B 0,C 180,E1 27401.189,E2 27401.189} C_VEL
LIN {X 0,Y 577.299,Z 420.266,A -85,B 0,C 180,E1 27400.897,E2 27400.897} C_VEL
LIN {X 0,Y 577.232,Z 420.29,A -85,B 0,C 180,E1 27397.948,E2 27397.948} C_VEL
LIN {X 0,Y 577.302,Z 420.266,A -85,B 0,C 180,E1 27394.817,E2 27394.817} C_VEL
LIN {X 0,Y 577.243,Z 420.294,A -85,B 0,C 180,E1 27391.733,E2 27391.733} C_VEL
LIN {X 0,Y 577.297,Z 420.256,A -85,B 0,C 180,E1 27388.557,E2 27388.557} C_VEL
LIN {X 0,Y 577.26,Z 420.325,A -85,B 0,C 180,E1 27385.519,E2 27385.519} C_VEL
LIN {X 0,Y 577.281,Z 420.321,A -85,B 0,C 180,E1 27382.185,E2 27382.185} C_VEL
LIN {X 0,Y 577.289,Z 420.308,A -85,B 0,C 180,E1 27379.109,E2 27379.109} C_VEL
LIN {X 0,Y 577.272,Z 420.298,A -85,B 0,C 180,E1 27375.883,E2 27375.883} C_VEL
LIN {X 0,Y 577.314,Z 420.31,A -85,B 0,C 180,E1 27372.809,E2 27372.809} C_VEL
LIN {X 0,Y 577.275,Z 420.319,A -85,B 0,C 180,E1 27369.572,E2 27369.572} C_VEL
LIN {X 0,Y 577.321,Z 420.297,A -85,B 0,C 180,E1 27366.364,E2 27366.364} C_VEL
LIN {X 0,Y 577.288,Z 420.311,A -85,B 0,C 180,E1 27363.177,E2 27363.177} C_VEL
LIN {X 0,Y 577.304,Z 420.313,A -85,B 0,C 180,E1 27359.802,E2 27359.802} C_VEL
LIN {X 0,Y 577.314,Z 420.297,A -85,B 0,C 180,E1 27356.525,E2 27356.525} C_VEL
LIN {X 0,Y 577.291,Z 420.303,A -85,B 0,C 180,E1 27353.236,E2 27353.236} C_VEL
LIN {X 0,Y 577.315,Z 420.315,A -85,B 0,C 180,E1 27350.026,E2 27350.026} C_VEL
LIN {X 0,Y 577.315,Z 420.303,A -85,B 0,C 180,E1 27346.682,E2 27346.682} C_VEL
LIN {X 0,Y 577.308,Z 420.297,A -85,B 0,C 180,E1 27343.395,E2 27343.395} C_VEL
LIN {X 0,Y 577.303,Z 420.311,A -85,B 0,C 180,E1 27340.133,E2 27340.133} C_VEL
LIN {X 0,Y 577.31,Z 420.304,A -85,B 0,C 180,E1 27336.849,E2 27336.849} C_VEL
LIN {X 0,Y 577.309,Z 420.288,A -85,B 0,C 180,E1 27333.565,E2 27333.565} C_VEL
LIN {X 0,Y 577.301,Z 420.313,A -85,B 0,C 180,E1 27330.192,E2 27330.192} C_VEL
LIN {X 0,Y 577.318,Z 420.315,A -85,B 0,C 180,E1 27326.936,E2 27326.936} C_VEL
LIN {X 0,Y 577.29,Z 420.304,A -85,B 0,C 180,E1 27323.649,E2 27323.649} C_VEL
LIN {X 0,Y 577.315,Z 420.295,A -85,B 0,C 180,E1 27320.404,E2 27320.404} C_VEL
LIN {X 0,Y 577.365,Z 420.606,A -85,B 0,C 180,E1 27318.581,E2 27318.581} C_VEL
LIN {X 0,Y 584.328,Z 436.973,A -85,B 0,C 180,E1 27316.088,E2 27316.088} C_VEL
LIN {X 0,Y 588.858,Z 447.813,A -85,B 0,C 180,E1 27314.576,E2 27314.576} C_VEL
LIN {X 0,Y 600.324,Z 466.222,A -85,B 0,C 180,E1 27313.153,E2 27313.153} C_VEL
LIN {X 0,Y 609.83,Z 482.982,A -85,B 0,C 180,E1 27312.034,E2 27312.034} C_VEL
LIN {X 0,Y 612.136,Z 494.978,A -85,B 0,C 180,E1 27311.647,E2 27311.647} C_VEL
LIN {X 0,Y 606.782,Z 731.117,A -85,B 0,C 180,E1 27308.479,E2 27308.479} C_VEL
LIN {X 0,Y 604.312,Z 841.013,A -85,B 0,C 180,E1 27307.001,E2 27307.001} C_VEL
LIN {X 0,Y 602.967,Z 866.903,A -85,B 0,C 180,E1 27306.495,E2 27306.495} C_VEL
LIN {X 0,Y 601.503,Z 888.401,A -85,B 0,C 180,E1 27305.927,E2 27305.927} C_VEL
LIN {X 0,Y 599.6,Z 912.332,A -85,B 0,C 180,E1 27305.122,E2 27305.122} C_VEL
LIN {X 0,Y 597.637,Z 933.188,A -85,B 0,C 180,E1 27304.259,E2 27304.259} C_VEL
LIN {X 0,Y 595.534,Z 953.982,A -85,B 0,C 180,E1 27303.249,E2 27303.249} C_VEL
LIN {X 0,Y 593.03,Z 976.197,A -85,B 0,C 180,E1 27301.967,E2 27301.967} C_VEL
LIN {X 0,Y 590.808,Z 995.409,A -85,B 0,C 180,E1 27300.687,E2 27300.687} C_VEL
LIN {X 0,Y 588.315,Z 1016.239,A -85,B 0,C 180,E1 27299.083,E2 27299.083} C_VEL
LIN {X 0,Y 586.246,Z 1033.289,A -85,B 0,C 180,E1 27297.585,E2 27297.585} C_VEL
LIN {X 0,Y 583.93,Z 1052.847,A -85,B 0,C 180,E1 27295.618,E2 27295.618} C_VEL
LIN {X 0,Y 582.216,Z 1067.7,A -85,B 0,C 180,E1 27293.91,E2 27293.91} C_VEL
LIN {X 0,Y 580.485,Z 1083.814,A -85,B 0,C 180,E1 27291.808,E2 27291.808} C_VEL
LIN {X 0,Y 579.191,Z 1096.62,A -85,B 0,C 180,E1 27289.883,E2 27289.883} C_VEL
LIN {X 0,Y 578.104,Z 1109.29,A -85,B 0,C 180,E1 27287.723,E2 27287.723} C_VEL
LIN {X 0,Y 577.249,Z 1120.445,A -85,B 0,C 180,E1 27285.471,E2 27285.471} C_VEL
LIN {X 0,Y 576.684,Z 1129.564,A -85,B 0,C 180,E1 27283.333,E2 27283.333} C_VEL
LIN {X 0,Y 576.264,Z 1137.906,A -85,B 0,C 180,E1 27280.902,E2 27280.902} C_VEL
LIN {X 0,Y 576.054,Z 1143.491,A -85,B 0,C 180,E1 27278.887,E2 27278.887} C_VEL
LIN {X 0,Y 575.953,Z 1148.695,A -85,B 0,C 180,E1 27276.479,E2 27276.479} C_VEL
LIN {X 0,Y 575.922,Z 1152.007,A -85,B 0,C 180,E1 27274.182,E2 27274.182} C_VEL
LIN {X 0,Y 575.91,Z 1153.902,A -85,B 0,C 180,E1 27271.99,E2 27271.99} C_VEL
LIN {X 0,Y 575.885,Z 1154.393,A -85,B 0,C 180,E1 27269.503,E2 27269.503} C_VEL
LIN {X 0,Y 575.893,Z 1153.493,A -85,B 0,C 180,E1 27267.413,E2 27267.413} C_VEL
LIN {X 0,Y 575.91,Z 1151.211,A -85,B 0,C 180,E1 27265.12,E2 27265.12} C_VEL
LIN {X 0,Y 575.974,Z 1147.308,A -85,B 0,C 180,E1 27262.82,E2 27262.82} C_VEL
LIN {X 0,Y 576.082,Z 1142.728,A -85,B 0,C 180,E1 27260.812,E2 27260.812} C_VEL
LIN {X 0,Y 576.336,Z 1136.069,A -85,B 0,C 180,E1 27258.491,E2 27258.491} C_VEL
LIN {X 0,Y 576.739,Z 1128.325,A -85,B 0,C 180,E1 27256.362,E2 27256.362} C_VEL
LIN {X 0,Y 577.311,Z 1119.518,A -85,B 0,C 180,E1 27254.324,E2 27254.324} C_VEL
LIN {X 0,Y 578.283,Z 1106.977,A -85,B 0,C 180,E1 27251.866,E2 27251.866} C_VEL
LIN {X 0,Y 579.324,Z 1095.35,A -85,B 0,C 180,E1 27249.912,E2 27249.912} C_VEL
LIN {X 0,Y 580.817,Z 1080.611,A -85,B 0,C 180,E1 27247.745,E2 27247.745} C_VEL
LIN {X 0,Y 582.414,Z 1066.022,A -85,B 0,C 180,E1 27245.883,E2 27245.883} C_VEL
LIN {X 0,Y 584.343,Z 1049.604,A -85,B 0,C 180,E1 27244.02,E2 27244.02} C_VEL
LIN {X 0,Y 586.509,Z 1031.305,A -85,B 0,C 180,E1 27242.227,E2 27242.227} C_VEL
LIN {X 0,Y 588.824,Z 1012.411,A -85,B 0,C 180,E1 27240.591,E2 27240.591} C_VEL
LIN {X 0,Y 591.137,Z 992.563,A -85,B 0,C 180,E1 27239.112,E2 27239.112} C_VEL
LIN {X 0,Y 593.425,Z 972.888,A -85,B 0,C 180,E1 27237.829,E2 27237.829} C_VEL
LIN {X 0,Y 595.792,Z 950.825,A -85,B 0,C 180,E1 27236.601,E2 27236.601} C_VEL
LIN {X 0,Y 597.704,Z 931.529,A -85,B 0,C 180,E1 27235.683,E2 27235.683} C_VEL
LIN {X 0,Y 599.794,Z 908.171,A -85,B 0,C 180,E1 27234.745,E2 27234.745} C_VEL
LIN {X 0,Y 601.497,Z 885.325,A -85,B 0,C 180,E1 27234.013,E2 27234.013} C_VEL
LIN {X 0,Y 603.097,Z 861.01,A -85,B 0,C 180,E1 27233.403,E2 27233.403} C_VEL
LIN {X 0,Y 604.146,Z 836.827,A -85,B 0,C 180,E1 27232.976,E2 27232.976} C_VEL
LIN {X 0,Y 608.969,Z 601.524,A -85,B 0,C 180,E1 27229.863,E2 27229.863} C_VEL
LIN {X 0,Y 611.131,Z 493.266,A -85,B 0,C 180,E1 27228.411,E2 27228.411} C_VEL
LIN {X 0,Y 608.335,Z 481.313,A -85,B 0,C 180,E1 27228.005,E2 27228.005} C_VEL
LIN {X 0,Y 591.765,Z 453.323,A -85,B 0,C 180,E1 27226.159,E2 27226.159} C_VEL
LIN {X 0,Y 588.684,Z 448.253,A -85,B 0,C 180,E1 27225.789,E2 27225.789} C_VEL
LIN {X 0,Y 581.508,Z 430.723,A -85,B 0,C 180,E1 27223.456,E2 27223.456} C_VEL
LIN {X 0,Y 577.31,Z 420.467,A -85,B 0,C 180,E1 27221.964,E2 27221.964} C_VEL
LIN {X 0,Y 577.319,Z 420.301,A -85,B 0,C 180,E1 27219.082,E2 27219.082} C_VEL
LIN {X 0,Y 577.295,Z 420.307,A -85,B 0,C 180,E1 27215.833,E2 27215.833} C_VEL
LIN {X 0,Y 577.301,Z 420.3,A -85,B 0,C 180,E1 27212.475,E2 27212.475} C_VEL
LIN {X 0,Y 577.314,Z 420.295,A -85,B 0,C 180,E1 27209.237,E2 27209.237} C_VEL
LIN {X 0,Y 577.3,Z 420.321,A -85,B 0,C 180,E1 27205.984,E2 27205.984} C_VEL
LIN {X 0,Y 577.314,Z 420.309,A -85,B 0,C 180,E1 27202.72,E2 27202.72} C_VEL
LIN {X 0,Y 577.313,Z 420.295,A -85,B 0,C 180,E1 27199.423,E2 27199.423} C_VEL
LIN {X 0,Y 577.311,Z 420.316,A -85,B 0,C 180,E1 27196.088,E2 27196.088} C_VEL
LIN {X 0,Y 577.301,Z 420.305,A -85,B 0,C 180,E1 27192.911,E2 27192.911} C_VEL
LIN {X 0,Y 577.309,Z 420.3,A -85,B 0,C 180,E1 27189.672,E2 27189.672} C_VEL
LIN {X 0,Y 577.306,Z 420.315,A -85,B 0,C 180,E1 27186.364,E2 27186.364} C_VEL
LIN {X 0,Y 577.296,Z 420.293,A -85,B 0,C 180,E1 27182.978,E2 27182.978} C_VEL
LIN {X 0,Y 577.319,Z 420.318,A -85,B 0,C 180,E1 27179.702,E2 27179.702} C_VEL
LIN {X 0,Y 577.285,Z 420.306,A -85,B 0,C 180,E1 27176.425,E2 27176.425} C_VEL
LIN {X 0,Y 577.312,Z 420.301,A -85,B 0,C 180,E1 27173.136,E2 27173.136} C_VEL
LIN {X 0,Y 577.31,Z 420.312,A -85,B 0,C 180,E1 27169.825,E2 27169.825} C_VEL
LIN {X 0,Y 577.271,Z 420.293,A -85,B 0,C 180,E1 27166.579,E2 27166.579} C_VEL
LIN {X 0,Y 577.323,Z 420.319,A -85,B 0,C 180,E1 27163.395,E2 27163.395} C_VEL
LIN {X 0,Y 577.265,Z 420.305,A -85,B 0,C 180,E1 27160.259,E2 27160.259} C_VEL
LIN {X 0,Y 577.313,Z 420.299,A -85,B 0,C 180,E1 27157.064,E2 27157.064} C_VEL
LIN {X 0,Y 577.268,Z 420.32,A -85,B 0,C 180,E1 27153.899,E2 27153.899} C_VEL
LIN {X 0,Y 577.265,Z 420.309,A -85,B 0,C 180,E1 27150.533,E2 27150.533} C_VEL
LIN {X 0,Y 577.269,Z 420.307,A -85,B 0,C 180,E1 27147.641,E2 27147.641} C_VEL
LIN {X 0,Y 577.249,Z 420.319,A -85,B 0,C 180,E1 27144.33,E2 27144.33} C_VEL
LIN {X 0,Y 577.307,Z 420.323,A -85,B 0,C 180,E1 27141.172,E2 27141.172} C_VEL
LIN {X 0,Y 577.224,Z 420.248,A -85,B 0,C 180,E1 27138.037,E2 27138.037} C_VEL
LIN {X 0,Y 577.299,Z 420.322,A -85,B 0,C 180,E1 27134.895,E2 27134.895} C_VEL
LIN {X 0,Y 577.262,Z 420.475,A -85,B 0,C 180,E1 27132.317,E2 27132.317} C_VEL
LIN {X 0,Y 577.604,Z 421.898,A -85,B 0,C 180,E1 27132.135,E2 27132.135} C_VEL
LIN {X 0,Y 579.557,Z 424.984,A -85,B 0,C 180,E1 27131.888,E2 27131.888} C_VEL
LIN {X 0,Y 580.877,Z 426.512,A -85,B 0,C 180,E1 27131.737,E2 27131.737} C_VEL
LIN {X 0,Y 583.627,Z 430.47,A -85,B 0,C 180,E1 27131.412,E2 27131.412} C_VEL
LIN {X 0,Y 598.334,Z 452.263,A -85,B 0,C 180,E1 27129.742,E2 27129.742} C_VEL
LIN {X 0,Y 611.466,Z 473.889,A -85,B 0,C 180,E1 27128.315,E2 27128.315} C_VEL
LIN {X 0,Y 608.406,Z 614.655,A -85,B 0,C 180,E1 27126.442,E2 27126.442} C_VEL
LIN {X 0,Y 607.481,Z 622.349,A -85,B 0,C 180,E1 27126.398,E2 27126.398} C_VEL
LIN {X 0,Y 602.147,Z 642.893,A -85,B 0,C 180,E1 27126.498,E2 27126.498} C_VEL
LIN {X 0,Y 601.397,Z 649.499,A -85,B 0,C 180,E1 27126.456,E2 27126.456} C_VEL
LIN {X 0,Y 597.877,Z 806.41,A -85,B 0,C 180,E1 27124.354,E2 27124.354} C_VEL
LIN {X 0,Y 596.673,Z 832.144,A -85,B 0,C 180,E1 27123.844,E2 27123.844} C_VEL
LIN {X 0,Y 595.344,Z 852.523,A -85,B 0,C 180,E1 27123.302,E2 27123.302} C_VEL
LIN {X 0,Y 593.65,Z 874.959,A -85,B 0,C 180,E1 27122.557,E2 27122.557} C_VEL
LIN {X 0,Y 591.576,Z 896.747,A -85,B 0,C 180,E1 27121.656,E2 27121.656} C_VEL
LIN {X 0,Y 589.645,Z 915.401,A -85,B 0,C 180,E1 27120.749,E2 27120.749} C_VEL
LIN {X 0,Y 587.008,Z 938.389,A -85,B 0,C 180,E1 27119.434,E2 27119.434} C_VEL
LIN {X 0,Y 584.66,Z 957.295,A -85,B 0,C 180,E1 27118.166,E2 27118.166} C_VEL
LIN {X 0,Y 582.04,Z 977.732,A -85,B 0,C 180,E1 27116.584,E2 27116.584} C_VEL
LIN {X 0,Y 579.723,Z 994.862,A -85,B 0,C 180,E1 27115.052,E2 27115.052} C_VEL
LIN {X 0,Y 577.372,Z 1012.567,A -85,B 0,C 180,E1 27113.257,E2 27113.257} C_VEL
LIN {X 0,Y 575.268,Z 1028.291,A -85,B 0,C 180,E1 27111.408,E2 27111.408} C_VEL
LIN {X 0,Y 573.43,Z 1043.014,A -85,B 0,C 180,E1 27109.454,E2 27109.454} C_VEL
LIN {X 0,Y 571.762,Z 1057.099,A -85,B 0,C 180,E1 27107.284,E2 27107.284} C_VEL
LIN {X 0,Y 570.554,Z 1068.675,A -85,B 0,C 180,E1 27105.241,E2 27105.241} C_VEL
LIN {X 0,Y 569.503,Z 1080.092,A -85,B 0,C 180,E1 27102.884,E2 27102.884} C_VEL
LIN {X 0,Y 568.843,Z 1088.902,A -85,B 0,C 180,E1 27100.738,E2 27100.738} C_VEL
LIN {X 0,Y 568.331,Z 1097.54,A -85,B 0,C 180,E1 27098.193,E2 27098.193} C_VEL
LIN {X 0,Y 568.071,Z 1103.583,A -85,B 0,C 180,E1 27095.961,E2 27095.961} C_VEL
LIN {X 0,Y 567.939,Z 1108.682,A -85,B 0,C 180,E1 27093.533,E2 27093.533} C_VEL
LIN {X 0,Y 567.901,Z 1111.875,A -85,B 0,C 180,E1 27091.312,E2 27091.312} C_VEL
LIN {X 0,Y 567.909,Z 1113.683,A -85,B 0,C 180,E1 27089.294,E2 27089.294} C_VEL
LIN {X 0,Y 567.903,Z 1114.488,A -85,B 0,C 180,E1 27086.871,E2 27086.871} C_VEL
LIN {X 0,Y 567.908,Z 1113.636,A -85,B 0,C 180,E1 27084.544,E2 27084.544} C_VEL
LIN {X 0,Y 567.905,Z 1111.782,A -85,B 0,C 180,E1 27082.514,E2 27082.514} C_VEL
LIN {X 0,Y 567.962,Z 1108.106,A -85,B 0,C 180,E1 27080.065,E2 27080.065} C_VEL
LIN {X 0,Y 568.096,Z 1102.964,A -85,B 0,C 180,E1 27077.704,E2 27077.704} C_VEL
LIN {X 0,Y 568.398,Z 1096.413,A -85,B 0,C 180,E1 27075.326,E2 27075.326} C_VEL
LIN {X 0,Y 568.904,Z 1087.985,A -85,B 0,C 180,E1 27072.931,E2 27072.931} C_VEL
LIN {X 0,Y 569.668,Z 1078.365,A -85,B 0,C 180,E1 27070.626,E2 27070.626} C_VEL
LIN {X 0,Y 570.675,Z 1067.302,A -85,B 0,C 180,E1 27068.411,E2 27068.411} C_VEL
LIN {X 0,Y 571.97,Z 1055.489,A -85,B 0,C 180,E1 27066.353,E2 27066.353} C_VEL
LIN {X 0,Y 573.684,Z 1040.96,A -85,B 0,C 180,E1 27064.168,E2 27064.168} C_VEL
LIN {X 0,Y 575.431,Z 1027.188,A -85,B 0,C 180,E1 27062.358,E2 27062.358} C_VEL
LIN {X 0,Y 577.783,Z 1009.397,A -85,B 0,C 180,E1 27060.313,E2 27060.313} C_VEL
LIN {X 0,Y 579.977,Z 993.247,A -85,B 0,C 180,E1 27058.699,E2 27058.699} C_VEL
LIN {X 0,Y 582.614,Z 973.718,A -85,B 0,C 180,E1 27056.982,E2 27056.982} C_VEL
LIN {X 0,Y 585.063,Z 954.829,A -85,B 0,C 180,E1 27055.55,E2 27055.55} C_VEL
LIN {X 0,Y 587.716,Z 934.071,A -85,B 0,C 180,E1 27054.179,E2 27054.179} C_VEL
LIN {X 0,Y 590.073,Z 913.317,A -85,B 0,C 180,E1 27053.018,E2 27053.018} C_VEL
LIN {X 0,Y 592.165,Z 893.706,A -85,B 0,C 180,E1 27052.075,E2 27052.075} C_VEL
LIN {X 0,Y 594.39,Z 869.332,A -85,B 0,C 180,E1 27051.105,E2 27051.105} C_VEL
LIN {X 0,Y 596.027,Z 848.195,A -85,B 0,C 180,E1 27050.426,E2 27050.426} C_VEL
LIN {X 0,Y 597.641,Z 822.085,A -85,B 0,C 180,E1 27049.786,E2 27049.786} C_VEL
LIN {X 0,Y 598.56,Z 800.16,A -85,B 0,C 180,E1 27049.401,E2 27049.401} C_VEL
LIN {X 0,Y 604.526,Z 550.124,A -85,B 0,C 180,E1 27046.025,E2 27046.025} C_VEL
LIN {X 0,Y 606.257,Z 476.939,A -85,B 0,C 180,E1 27045.019,E2 27045.019} C_VEL
LIN {X 0,Y 593.909,Z 456.829,A -85,B 0,C 180,E1 27043.552,E2 27043.552} C_VEL
LIN {X 0,Y 579.978,Z 436.988,A -85,B 0,C 180,E1 27041.818,E2 27041.818} C_VEL
LIN {X 0,Y 575.862,Z 431.498,A -85,B 0,C 180,E1 27041.285,E2 27041.285} C_VEL
LIN {X 0,Y 573.253,Z 427.602,A -85,B 0,C 180,E1 27040.934,E2 27040.934} C_VEL
LIN {X 0,Y 570.07,Z 423.797,A -85,B 0,C 180,E1 27040.514,E2 27040.514} C_VEL
LIN {X 0,Y 569.414,Z 421.936,A -85,B 0,C 180,E1 27040.35,E2 27040.35} C_VEL
LIN {X 0,Y 569.29,Z 421.278,A -85,B 0,C 180,E1 27040.004,E2 27040.004} C_VEL
LIN {X 0,Y 569.355,Z 421.242,A -85,B 0,C 180,E1 27037.04,E2 27037.04} C_VEL
LIN {X 0,Y 569.303,Z 421.299,A -85,B 0,C 180,E1 27033.824,E2 27033.824} C_VEL
LIN {X 0,Y 569.358,Z 421.237,A -85,B 0,C 180,E1 27030.617,E2 27030.617} C_VEL
LIN {X 0,Y 569.313,Z 421.28,A -85,B 0,C 180,E1 27027.624,E2 27027.624} C_VEL
LIN {X 0,Y 569.353,Z 421.289,A -85,B 0,C 180,E1 27024.375,E2 27024.375} C_VEL
LIN {X 0,Y 569.333,Z 421.305,A -85,B 0,C 180,E1 27021.318,E2 27021.318} C_VEL
LIN {X 0,Y 569.335,Z 421.31,A -85,B 0,C 180,E1 27017.899,E2 27017.899} C_VEL
LIN {X 0,Y 569.385,Z 421.292,A -85,B 0,C 180,E1 27014.752,E2 27014.752} C_VEL
LIN {X 0,Y 569.333,Z 421.289,A -85,B 0,C 180,E1 27011.481,E2 27011.481} C_VEL
LIN {X 0,Y 569.377,Z 421.298,A -85,B 0,C 180,E1 27008.178,E2 27008.178} C_VEL
LIN {X 0,Y 569.363,Z 421.304,A -85,B 0,C 180,E1 27004.937,E2 27004.937} C_VEL
LIN {X 0,Y 569.348,Z 421.283,A -85,B 0,C 180,E1 27001.61,E2 27001.61} C_VEL
LIN {X 0,Y 569.377,Z 421.29,A -85,B 0,C 180,E1 26998.39,E2 26998.39} C_VEL
LIN {X 0,Y 569.358,Z 421.304,A -85,B 0,C 180,E1 26995.063,E2 26995.063} C_VEL
LIN {X 0,Y 569.373,Z 421.288,A -85,B 0,C 180,E1 26991.72,E2 26991.72} C_VEL
LIN {X 0,Y 569.372,Z 421.286,A -85,B 0,C 180,E1 26988.451,E2 26988.451} C_VEL
LIN {X 0,Y 569.362,Z 421.309,A -85,B 0,C 180,E1 26985.143,E2 26985.143} C_VEL
LIN {X 0,Y 569.373,Z 421.304,A -85,B 0,C 180,E1 26981.818,E2 26981.818} C_VEL
LIN {X 0,Y 569.374,Z 421.273,A -85,B 0,C 180,E1 26978.467,E2 26978.467} C_VEL
LIN {X 0,Y 569.377,Z 421.307,A -85,B 0,C 180,E1 26975.184,E2 26975.184} C_VEL
LIN {X 0,Y 569.358,Z 421.293,A -85,B 0,C 180,E1 26971.923,E2 26971.923} C_VEL
LIN {X 0,Y 569.376,Z 421.278,A -85,B 0,C 180,E1 26968.68,E2 26968.68} C_VEL
LIN {X 0,Y 569.365,Z 421.293,A -85,B 0,C 180,E1 26965.442,E2 26965.442} C_VEL
LIN {X 0,Y 569.352,Z 421.302,A -85,B 0,C 180,E1 26962.049,E2 26962.049} C_VEL
LIN {X 0,Y 569.378,Z 421.468,A -85,B 0,C 180,E1 26959.412,E2 26959.412} C_VEL
LIN {X 0,Y 571.02,Z 425.285,A -85,B 0,C 180,E1 26958.755,E2 26958.755} C_VEL
LIN {X 0,Y 577.822,Z 441.05,A -85,B 0,C 180,E1 26956.33,E2 26956.33} C_VEL
LIN {X 0,Y 580.543,Z 447.383,A -85,B 0,C 180,E1 26955.424,E2 26955.424} C_VEL
LIN {X 0,Y 592.828,Z 467.047,A -85,B 0,C 180,E1 26953.842,E2 26953.842} C_VEL
LIN {X 0,Y 604.297,Z 486.624,A -85,B 0,C 180,E1 26952.464,E2 26952.464} C_VEL
LIN {X 0,Y 606.19,Z 496.861,A -85,B 0,C 180,E1 26952.133,E2 26952.133} C_VEL
LIN {X 0,Y 600.556,Z 732.253,A -85,B 0,C 180,E1 26948.947,E2 26948.947} C_VEL
LIN {X 0,Y 597.983,Z 840.784,A -85,B 0,C 180,E1 26947.473,E2 26947.473} C_VEL
LIN {X 0,Y 596.555,Z 866.835,A -85,B 0,C 180,E1 26946.96,E2 26946.96} C_VEL
LIN {X 0,Y 595.004,Z 888.5,A -85,B 0,C 180,E1 26946.382,E2 26946.382} C_VEL
LIN {X 0,Y 592.877,Z 913.599,A -85,B 0,C 180,E1 26945.521,E2 26945.521} C_VEL
LIN {X 0,Y 590.877,Z 933.782,A -85,B 0,C 180,E1 26944.672,E2 26944.672} C_VEL
LIN {X 0,Y 588.505,Z 955.908,A -85,B 0,C 180,E1 26943.576,E2 26943.576} C_VEL
LIN {X 0,Y 586.001,Z 976.758,A -85,B 0,C 180,E1 26942.345,E2 26942.345} C_VEL
LIN {X 0,Y 583.475,Z 997.486,A -85,B 0,C 180,E1 26940.938,E2 26940.938} C_VEL
LIN {X 0,Y 580.936,Z 1017.191,A -85,B 0,C 180,E1 26939.376,E2 26939.376} C_VEL
LIN {X 0,Y 578.667,Z 1034.916,A -85,B 0,C 180,E1 26937.785,E2 26937.785} C_VEL
LIN {X 0,Y 576.328,Z 1053.481,A -85,B 0,C 180,E1 26935.87,E2 26935.87} C_VEL
LIN {X 0,Y 574.53,Z 1068.254,A -85,B 0,C 180,E1 26934.141,E2 26934.141} C_VEL
LIN {X 0,Y 572.648,Z 1084.699,A -85,B 0,C 180,E1 26931.942,E2 26931.942} C_VEL
LIN {X 0,Y 571.29,Z 1097.534,A -85,B 0,C 180,E1 26929.969,E2 26929.969} C_VEL
LIN {X 0,Y 570.049,Z 1111.104,A -85,B 0,C 180,E1 26927.56,E2 26927.56} C_VEL
LIN {X 0,Y 569.267,Z 1121.083,A -85,B 0,C 180,E1 26925.485,E2 26925.485} C_VEL
LIN {X 0,Y 568.649,Z 1130.849,A -85,B 0,C 180,E1 26923.111,E2 26923.111} C_VEL
LIN {X 0,Y 568.266,Z 1138.387,A -85,B 0,C 180,E1 26920.852,E2 26920.852} C_VEL
LIN {X 0,Y 568.051,Z 1144.506,A -85,B 0,C 180,E1 26918.605,E2 26918.605} C_VEL
LIN {X 0,Y 567.954,Z 1149.333,A -85,B 0,C 180,E1 26916.165,E2 26916.165} C_VEL
LIN {X 0,Y 567.919,Z 1152.234,A -85,B 0,C 180,E1 26914.038,E2 26914.038} C_VEL
LIN {X 0,Y 567.898,Z 1154.144,A -85,B 0,C 180,E1 26911.614,E2 26911.614} C_VEL
LIN {X 0,Y 567.886,Z 1154.348,A -85,B 0,C 180,E1 26909.294,E2 26909.294} C_VEL
LIN {X 0,Y 567.888,Z 1153.425,A -85,B 0,C 180,E1 26907.275,E2 26907.275} C_VEL
LIN {X 0,Y 567.905,Z 1150.929,A -85,B 0,C 180,E1 26904.848,E2 26904.848} C_VEL
LIN {X 0,Y 567.972,Z 1147.101,A -85,B 0,C 180,E1 26902.616,E2 26902.616} C_VEL
LIN {X 0,Y 568.103,Z 1142.694,A -85,B 0,C 180,E1 26900.681,E2 26900.681} C_VEL
LIN {X 0,Y 568.37,Z 1135.894,A -85,B 0,C 180,E1 26898.328,E2 26898.328} C_VEL
LIN {X 0,Y 568.828,Z 1127.383,A -85,B 0,C 180,E1 26896.005,E2 26896.005} C_VEL
LIN {X 0,Y 569.469,Z 1118.293,A -85,B 0,C 180,E1 26893.894,E2 26893.894} C_VEL
LIN {X 0,Y 570.48,Z 1106.102,A -85,B 0,C 180,E1 26891.504,E2 26891.504} C_VEL
LIN {X 0,Y 571.631,Z 1094.413,A -85,B 0,C 180,E1 26889.522,E2 26889.522} C_VEL
LIN {X 0,Y 573.32,Z 1078.755,A -85,B 0,C 180,E1 26887.221,E2 26887.221} C_VEL
LIN {X 0,Y 574.942,Z 1064.872,A -85,B 0,C 180,E1 26885.44,E2 26885.44} C_VEL
LIN {X 0,Y 577.129,Z 1047.271,A -85,B 0,C 180,E1 26883.449,E2 26883.449} C_VEL
LIN {X 0,Y 579.283,Z 1030.248,A -85,B 0,C 180,E1 26881.774,E2 26881.774} C_VEL
LIN {X 0,Y 581.752,Z 1011.006,A -85,B 0,C 180,E1 26880.103,E2 26880.103} C_VEL
LIN {X 0,Y 584.163,Z 991.454,A -85,B 0,C 180,E1 26878.644,E2 26878.644} C_VEL
LIN {X 0,Y 586.692,Z 970.84,A -85,B 0,C 180,E1 26877.299,E2 26877.299} C_VEL
LIN {X 0,Y 589.063,Z 949.235,A -85,B 0,C 180,E1 26876.103,E2 26876.103} C_VEL
LIN {X 0,Y 591.079,Z 929.879,A -85,B 0,C 180,E1 26875.185,E2 26875.185} C_VEL
LIN {X 0,Y 593.372,Z 904.576,A -85,B 0,C 180,E1 26874.186,E2 26874.186} C_VEL
LIN {X 0,Y 595.078,Z 882.927,A -85,B 0,C 180,E1 26873.504,E2 26873.504} C_VEL
LIN {X 0,Y 596.796,Z 856.769,A -85,B 0,C 180,E1 26872.875,E2 26872.875} C_VEL
LIN {X 0,Y 597.738,Z 834.883,A -85,B 0,C 180,E1 26872.496,E2 26872.496} C_VEL
LIN {X 0,Y 602.769,Z 600.481,A -85,B 0,C 180,E1 26869.37,E2 26869.37} C_VEL
LIN {X 0,Y 604.999,Z 495.065,A -85,B 0,C 180,E1 26867.944,E2 26867.944} C_VEL
LIN {X 0,Y 602.762,Z 485.558,A -85,B 0,C 180,E1 26867.613,E2 26867.613} C_VEL
LIN {X 0,Y 587.075,Z 458.839,A -85,B 0,C 180,E1 26865.828,E2 26865.828} C_VEL
LIN {X 0,Y 580.117,Z 447.512,A -85,B 0,C 180,E1 26864.965,E2 26864.965} C_VEL
LIN {X 0,Y 572.374,Z 428.688,A -85,B 0,C 180,E1 26862.358,E2 26862.358} C_VEL
LIN {X 0,Y 569.407,Z 421.447,A -85,B 0,C 180,E1 26861.254,E2 26861.254} C_VEL
LIN {X 0,Y 569.35,Z 421.309,A -85,B 0,C 180,E1 26858.056,E2 26858.056} C_VEL
LIN {X 0,Y 569.374,Z 421.31,A -85,B 0,C 180,E1 26854.68,E2 26854.68} C_VEL
LIN {X 0,Y 569.379,Z 421.305,A -85,B 0,C 180,E1 26851.32,E2 26851.32} C_VEL
LIN {X 0,Y 569.355,Z 421.286,A -85,B 0,C 180,E1 26848.077,E2 26848.077} C_VEL
LIN {X 0,Y 569.373,Z 421.283,A -85,B 0,C 180,E1 26844.78,E2 26844.78} C_VEL
LIN {X 0,Y 569.381,Z 421.309,A -85,B 0,C 180,E1 26841.424,E2 26841.424} C_VEL
LIN {X 0,Y 569.366,Z 421.293,A -85,B 0,C 180,E1 26838.004,E2 26838.004} C_VEL
LIN {X 0,Y 569.364,Z 421.285,A -85,B 0,C 180,E1 26834.752,E2 26834.752} C_VEL
LIN {X 0,Y 569.376,Z 421.309,A -85,B 0,C 180,E1 26831.446,E2 26831.446} C_VEL
LIN {X 0,Y 569.378,Z 421.28,A -85,B 0,C 180,E1 26828.076,E2 26828.076} C_VEL
LIN {X 0,Y 569.355,Z 421.298,A -85,B 0,C 180,E1 26824.836,E2 26824.836} C_VEL
LIN {X 0,Y 569.378,Z 421.294,A -85,B 0,C 180,E1 26821.509,E2 26821.509} C_VEL
LIN {X 0,Y 569.355,Z 421.288,A -85,B 0,C 180,E1 26818.289,E2 26818.289} C_VEL
LIN {X 0,Y 569.352,Z 421.31,A -85,B 0,C 180,E1 26814.861,E2 26814.861} C_VEL
LIN {X 0,Y 569.38,Z 421.276,A -85,B 0,C 180,E1 26811.619,E2 26811.619} C_VEL
LIN {X 0,Y 569.337,Z 421.306,A -85,B 0,C 180,E1 26808.348,E2 26808.348} C_VEL
LIN {X 0,Y 569.367,Z 421.291,A -85,B 0,C 180,E1 26805.039,E2 26805.039} C_VEL
LIN {X 0,Y 569.351,Z 421.29,A -85,B 0,C 180,E1 26801.824,E2 26801.824} C_VEL
LIN {X 0,Y 569.331,Z 421.311,A -85,B 0,C 180,E1 26798.563,E2 26798.563} C_VEL
LIN {X 0,Y 569.375,Z 421.28,A -85,B 0,C 180,E1 26795.405,E2 26795.405} C_VEL
LIN {X 0,Y 569.317,Z 421.298,A -85,B 0,C 180,E1 26792.262,E2 26792.262} C_VEL
LIN {X 0,Y 569.386,Z 421.308,A -85,B 0,C 180,E1 26789.151,E2 26789.151} C_VEL
LIN {X 0,Y 569.31,Z 421.308,A -85,B 0,C 180,E1 26785.926,E2 26785.926} C_VEL
LIN {X 0,Y 569.337,Z 421.294,A -85,B 0,C 180,E1 26782.706,E2 26782.706} C_VEL
LIN {X 0,Y 569.298,Z 421.275,A -85,B 0,C 180,E1 26779.82,E2 26779.82} C_VEL
LIN {X 0,Y 569.322,Z 421.244,A -85,B 0,C 180,E1 26776.63,E2 26776.63} C_VEL
LIN {X 0,Y 569.287,Z 421.278,A -85,B 0,C 180,E1 26773.79,E2 26773.79} C_VEL
LIN {X 0,Y 569.386,Z 421.561,A -85,B 0,C 180,E1 26773.069,E2 26773.069} C_VEL
LIN {X 0,Y 569.834,Z 423.161,A -85,B 0,C 180,E1 26772.877,E2 26772.877} C_VEL
LIN {X 0,Y 571.951,Z 426.239,A -85,B 0,C 180,E1 26772.608,E2 26772.608} C_VEL
LIN {X 0,Y 573.137,Z 427.851,A -85,B 0,C 180,E1 26772.463,E2 26772.463} C_VEL
LIN {X 0,Y 575.956,Z 431.734,A -85,B 0,C 180,E1 26772.121,E2 26772.121} C_VEL
LIN {X 0,Y 592.801,Z 456.513,A -85,B 0,C 180,E1 26770.155,E2 26770.155} C_VEL
LIN {X 0,Y 605.326,Z 477.201,A -85,B 0,C 180,E1 26768.766,E2 26768.766} C_VEL
LIN {X 0,Y 601.397,Z 649.499,A -85,B 0,C 180,E1 26766.456,E2 26766.456} C_VEL
LIN {X 0,Y 600.436,Z 657.193,A -85,B 0,C 180,E1 26766.414,E2 26766.414} C_VEL
LIN {X 0,Y 595.106,Z 677.731,A -85,B 0,C 180,E1 26766.515,E2 26766.515} C_VEL
LIN {X 0,Y 594.357,Z 684.334,A -85,B 0,C 180,E1 26766.473,E2 26766.473} C_VEL
LIN {X 0,Y 591.455,Z 807.033,A -85,B 0,C 180,E1 26764.81,E2 26764.81} C_VEL
LIN {X 0,Y 590.206,Z 832.519,A -85,B 0,C 180,E1 26764.299,E2 26764.299} C_VEL
LIN {X 0,Y 588.816,Z 853,A -85,B 0,C 180,E1 26763.749,E2 26763.749} C_VEL
LIN {X 0,Y 586.985,Z 876.041,A -85,B 0,C 180,E1 26762.973,E2 26762.973} C_VEL
LIN {X 0,Y 584.83,Z 897.734,A -85,B 0,C 180,E1 26762.064,E2 26762.064} C_VEL
LIN {X 0,Y 582.711,Z 917.317,A -85,B 0,C 180,E1 26761.098,E2 26761.098} C_VEL
LIN {X 0,Y 579.958,Z 939.999,A -85,B 0,C 180,E1 26759.771,E2 26759.771} C_VEL
LIN {X 0,Y 577.495,Z 959.001,A -85,B 0,C 180,E1 26758.474,E2 26758.474} C_VEL
LIN {X 0,Y 574.6,Z 980.273,A -85,B 0,C 180,E1 26756.785,E2 26756.785} C_VEL
LIN {X 0,Y 572.292,Z 996.66,A -85,B 0,C 180,E1 26755.289,E2 26755.289} C_VEL
LIN {X 0,Y 569.704,Z 1015.039,A -85,B 0,C 180,E1 26753.369,E2 26753.369} C_VEL
LIN {X 0,Y 567.643,Z 1029.753,A -85,B 0,C 180,E1 26751.602,E2 26751.602} C_VEL
LIN {X 0,Y 565.634,Z 1045.056,A -85,B 0,C 180,E1 26749.518,E2 26749.518} C_VEL
LIN {X 0,Y 563.979,Z 1058.204,A -85,B 0,C 180,E1 26747.435,E2 26747.435} C_VEL
LIN {X 0,Y 562.601,Z 1070.86,A -85,B 0,C 180,E1 26745.145,E2 26745.145} C_VEL
LIN {X 0,Y 561.558,Z 1081.463,A -85,B 0,C 180,E1 26742.86,E2 26742.86} C_VEL
LIN {X 0,Y 560.854,Z 1090.538,A -85,B 0,C 180,E1 26740.581,E2 26740.581} C_VEL
LIN {X 0,Y 560.362,Z 1098.247,A -85,B 0,C 180,E1 26738.207,E2 26738.207} C_VEL
LIN {X 0,Y 560.098,Z 1103.946,A -85,B 0,C 180,E1 26736.046,E2 26736.046} C_VEL
LIN {X 0,Y 559.95,Z 1108.97,A -85,B 0,C 180,E1 26733.583,E2 26733.583} C_VEL
LIN {X 0,Y 559.905,Z 1112.07,A -85,B 0,C 180,E1 26731.33,E2 26731.33} C_VEL
LIN {X 0,Y 559.91,Z 1113.818,A -85,B 0,C 180,E1 26729.284,E2 26729.284} C_VEL
LIN {X 0,Y 559.897,Z 1114.546,A -85,B 0,C 180,E1 26726.724,E2 26726.724} C_VEL
LIN {X 0,Y 559.908,Z 1113.717,A -85,B 0,C 180,E1 26724.466,E2 26724.466} C_VEL
LIN {X 0,Y 559.929,Z 1111.775,A -85,B 0,C 180,E1 26722.303,E2 26722.303} C_VEL
LIN {X 0,Y 560,Z 1107.782,A -85,B 0,C 180,E1 26719.681,E2 26719.681} C_VEL
LIN {X 0,Y 560.137,Z 1103.139,A -85,B 0,C 180,E1 26717.526,E2 26717.526} C_VEL
LIN {X 0,Y 560.474,Z 1096.564,A -85,B 0,C 180,E1 26715.114,E2 26715.114} C_VEL
LIN {X 0,Y 560.994,Z 1088.506,A -85,B 0,C 180,E1 26712.79,E2 26712.79} C_VEL
LIN {X 0,Y 561.759,Z 1079.373,A -85,B 0,C 180,E1 26710.558,E2 26710.558} C_VEL
LIN {X 0,Y 562.881,Z 1067.918,A -85,B 0,C 180,E1 26708.206,E2 26708.206} C_VEL
LIN {X 0,Y 564.216,Z 1056.423,A -85,B 0,C 180,E1 26706.168,E2 26706.168} C_VEL
LIN {X 0,Y 566.07,Z 1041.69,A -85,B 0,C 180,E1 26703.907,E2 26703.907} C_VEL
LIN {X 0,Y 567.91,Z 1027.96,A -85,B 0,C 180,E1 26702.074,E2 26702.074} C_VEL
LIN {X 0,Y 570.37,Z 1010.467,A -85,B 0,C 180,E1 26700.025,E2 26700.025} C_VEL
LIN {X 0,Y 572.729,Z 994.048,A -85,B 0,C 180,E1 26698.355,E2 26698.355} C_VEL
LIN {X 0,Y 575.463,Z 974.975,A -85,B 0,C 180,E1 26696.646,E2 26696.646} C_VEL
LIN {X 0,Y 578.041,Z 956.098,A -85,B 0,C 180,E1 26695.192,E2 26695.192} C_VEL
LIN {X 0,Y 580.819,Z 935.543,A -85,B 0,C 180,E1 26693.809,E2 26693.809} C_VEL
LIN {X 0,Y 583.396,Z 913.975,A -85,B 0,C 180,E1 26692.585,E2 26692.585} C_VEL
LIN {X 0,Y 585.584,Z 894.425,A -85,B 0,C 180,E1 26691.634,E2 26691.634} C_VEL
LIN {X 0,Y 587.906,Z 870.276,A -85,B 0,C 180,E1 26690.66,E2 26690.66} C_VEL
LIN {X 0,Y 589.652,Z 848.74,A -85,B 0,C 180,E1 26689.96,E2 26689.96} C_VEL
LIN {X 0,Y 591.358,Z 822.444,A -85,B 0,C 180,E1 26689.309,E2 26689.309} C_VEL
LIN {X 0,Y 592.318,Z 800.45,A -85,B 0,C 180,E1 26688.919,E2 26688.919} C_VEL
LIN {X 0,Y 598.589,Z 550.639,A -85,B 0,C 180,E1 26685.516,E2 26685.516} C_VEL
LIN {X 0,Y 600.343,Z 480.307,A -85,B 0,C 180,E1 26684.541,E2 26684.541} C_VEL
LIN {X 0,Y 588.496,Z 461.048,A -85,B 0,C 180,E1 26683.097,E2 26683.097} C_VEL
LIN {X 0,Y 575.669,Z 442.844,A -85,B 0,C 180,E1 26681.468,E2 26681.468} C_VEL
LIN {X 0,Y 569.074,Z 433.563,A -85,B 0,C 180,E1 26680.583,E2 26680.583} C_VEL
LIN {X 0,Y 565.922,Z 429.696,A -85,B 0,C 180,E1 26680.158,E2 26680.158} C_VEL
LIN {X 0,Y 564.762,Z 427.874,A -85,B 0,C 180,E1 26679.992,E2 26679.992} C_VEL
LIN {X 0,Y 562.36,Z 425.266,A -85,B 0,C 180,E1 26679.666,E2 26679.666} C_VEL
LIN {X 0,Y 561.504,Z 423.036,A -85,B 0,C 180,E1 26679.474,E2 26679.474} C_VEL
LIN {X 0,Y 561.407,Z 422.328,A -85,B 0,C 180,E1 26679.217,E2 26679.217} C_VEL
LIN {X 0,Y 561.355,Z 422.228,A -85,B 0,C 180,E1 26676.001,E2 26676.001} C_VEL
LIN {X 0,Y 561.432,Z 422.296,A -85,B 0,C 180,E1 26672.78,E2 26672.78} C_VEL
LIN {X 0,Y 561.366,Z 422.22,A -85,B 0,C 180,E1 26669.632,E2 26669.632} C_VEL
LIN {X 0,Y 561.406,Z 422.301,A -85,B 0,C 180,E1 26666.326,E2 26666.326} C_VEL
LIN {X 0,Y 561.404,Z 422.286,A -85,B 0,C 180,E1 26663.18,E2 26663.18} C_VEL
LIN {X 0,Y 561.389,Z 422.279,A -85,B 0,C 180,E1 26659.877,E2 26659.877} C_VEL
LIN {X 0,Y 561.443,Z 422.275,A -85,B 0,C 180,E1 26656.636,E2 26656.636} C_VEL
LIN {X 0,Y 561.397,Z 422.301,A -85,B 0,C 180,E1 26653.388,E2 26653.388} C_VEL
LIN {X 0,Y 561.422,Z 422.292,A -85,B 0,C 180,E1 26650.052,E2 26650.052} C_VEL
LIN {X 0,Y 561.441,Z 422.272,A -85,B 0,C 180,E1 26646.75,E2 26646.75} C_VEL
LIN {X 0,Y 561.406,Z 422.295,A -85,B 0,C 180,E1 26643.472,E2 26643.472} C_VEL
LIN {X 0,Y 561.447,Z 422.29,A -85,B 0,C 180,E1 26640.102,E2 26640.102} C_VEL
LIN {X 0,Y 561.431,Z 422.27,A -85,B 0,C 180,E1 26636.733,E2 26636.733} C_VEL
LIN {X 0,Y 561.415,Z 422.28,A -85,B 0,C 180,E1 26633.352,E2 26633.352} C_VEL
LIN {X 0,Y 561.438,Z 422.293,A -85,B 0,C 180,E1 26630.02,E2 26630.02} C_VEL
LIN {X 0,Y 561.439,Z 422.281,A -85,B 0,C 180,E1 26626.613,E2 26626.613} C_VEL
LIN {X 0,Y 561.425,Z 422.273,A -85,B 0,C 180,E1 26623.231,E2 26623.231} C_VEL
LIN {X 0,Y 561.426,Z 422.287,A -85,B 0,C 180,E1 26620.004,E2 26620.004} C_VEL
LIN {X 0,Y 561.439,Z 422.284,A -85,B 0,C 180,E1 26616.6,E2 26616.6} C_VEL
LIN {X 0,Y 561.435,Z 422.261,A -85,B 0,C 180,E1 26613.219,E2 26613.219} C_VEL
LIN {X 0,Y 561.417,Z 422.287,A -85,B 0,C 180,E1 26609.949,E2 26609.949} C_VEL
LIN {X 0,Y 561.441,Z 422.298,A -85,B 0,C 180,E1 26606.612,E2 26606.612} C_VEL
LIN {X 0,Y 561.434,Z 422.285,A -85,B 0,C 180,E1 26603.244,E2 26603.244} C_VEL
LIN {X 0,Y 561.452,Z 422.482,A -85,B 0,C 180,E1 26600.232,E2 26600.232} C_VEL
LIN {X 0,Y 562.983,Z 426.165,A -85,B 0,C 180,E1 26599.589,E2 26599.589} C_VEL
LIN {X 0,Y 570.15,Z 442.474,A -85,B 0,C 180,E1 26596.984,E2 26596.984} C_VEL
LIN {X 0,Y 572.022,Z 446.932,A -85,B 0,C 180,E1 26596.333,E2 26596.333} C_VEL
LIN {X 0,Y 584.462,Z 466.283,A -85,B 0,C 180,E1 26594.673,E2 26594.673} C_VEL
LIN {X 0,Y 596.853,Z 487.182,A -85,B 0,C 180,E1 26593.131,E2 26593.131} C_VEL
LIN {X 0,Y 599.096,Z 491.642,A -85,B 0,C 180,E1 26592.852,E2 26592.852} C_VEL
LIN {X 0,Y 600.289,Z 498.675,A -85,B 0,C 180,E1 26592.63,E2 26592.63} C_VEL
LIN {X 0,Y 594.37,Z 733.706,A -85,B 0,C 180,E1 26589.421,E2 26589.421} C_VEL
LIN {X 0,Y 591.701,Z 840.515,A -85,B 0,C 180,E1 26587.956,E2 26587.956} C_VEL
LIN {X 0,Y 590.204,Z 866.547,A -85,B 0,C 180,E1 26587.44,E2 26587.44} C_VEL
LIN {X 0,Y 588.565,Z 888.374,A -85,B 0,C 180,E1 26586.854,E2 26586.854} C_VEL
LIN {X 0,Y 586.315,Z 913.612,A -85,B 0,C 180,E1 26585.98,E2 26585.98} C_VEL
LIN {X 0,Y 584.275,Z 933.256,A -85,B 0,C 180,E1 26585.147,E2 26585.147} C_VEL
LIN {X 0,Y 581.729,Z 955.808,A -85,B 0,C 180,E1 26584.02,E2 26584.02} C_VEL
LIN {X 0,Y 579.069,Z 976.859,A -85,B 0,C 180,E1 26582.763,E2 26582.763} C_VEL
LIN {X 0,Y 576.425,Z 997.314,A -85,B 0,C 180,E1 26581.359,E2 26581.359} C_VEL
LIN {X 0,Y 573.749,Z 1016.971,A -85,B 0,C 180,E1 26579.781,E2 26579.781} C_VEL
LIN {X 0,Y 571.387,Z 1034.409,A -85,B 0,C 180,E1 26578.196,E2 26578.196} C_VEL
LIN {X 0,Y 568.86,Z 1053.179,A -85,B 0,C 180,E1 26576.236,E2 26576.236} C_VEL
LIN {X 0,Y 566.957,Z 1067.949,A -85,B 0,C 180,E1 26574.485,E2 26574.485} C_VEL
LIN {X 0,Y 564.929,Z 1084.584,A -85,B 0,C 180,E1 26572.228,E2 26572.228} C_VEL
LIN {X 0,Y 563.509,Z 1097.309,A -85,B 0,C 180,E1 26570.243,E2 26570.243} C_VEL
LIN {X 0,Y 562.192,Z 1110.806,A -85,B 0,C 180,E1 26567.813,E2 26567.813} C_VEL
LIN {X 0,Y 561.35,Z 1120.786,A -85,B 0,C 180,E1 26565.709,E2 26565.709} C_VEL
LIN {X 0,Y 560.691,Z 1130.554,A -85,B 0,C 180,E1 26563.3,E2 26563.3} C_VEL
LIN {X 0,Y 560.28,Z 1138.095,A -85,B 0,C 180,E1 26561.009,E2 26561.009} C_VEL
LIN {X 0,Y 560.053,Z 1144.221,A -85,B 0,C 180,E1 26558.729,E2 26558.729} C_VEL
LIN {X 0,Y 559.954,Z 1149.156,A -85,B 0,C 180,E1 26556.253,E2 26556.253} C_VEL
LIN {X 0,Y 559.921,Z 1152.125,A -85,B 0,C 180,E1 26554.096,E2 26554.096} C_VEL
LIN {X 0,Y 559.899,Z 1154.076,A -85,B 0,C 180,E1 26551.637,E2 26551.637} C_VEL
LIN {X 0,Y 559.885,Z 1154.31,A -85,B 0,C 180,E1 26549.386,E2 26549.386} C_VEL
LIN {X 0,Y 559.89,Z 1153.412,A -85,B 0,C 180,E1 26547.339,E2 26547.339} C_VEL
LIN {X 0,Y 559.907,Z 1151.075,A -85,B 0,C 180,E1 26544.98,E2 26544.98} C_VEL
LIN {X 0,Y 559.972,Z 1147.087,A -85,B 0,C 180,E1 26542.613,E2 26542.613} C_VEL
LIN {X 0,Y 560.12,Z 1142.408,A -85,B 0,C 180,E1 26540.547,E2 26540.547} C_VEL
LIN {X 0,Y 560.403,Z 1135.606,A -85,B 0,C 180,E1 26538.159,E2 26538.159} C_VEL
LIN {X 0,Y 560.873,Z 1127.335,A -85,B 0,C 180,E1 26535.863,E2 26535.863} C_VEL
LIN {X 0,Y 561.53,Z 1118.471,A -85,B 0,C 180,E1 26533.766,E2 26533.766} C_VEL
LIN {X 0,Y 562.61,Z 1106.221,A -85,B 0,C 180,E1 26531.311,E2 26531.311} C_VEL
LIN {X 0,Y 563.804,Z 1094.766,A -85,B 0,C 180,E1 26529.334,E2 26529.334} C_VEL
LIN {X 0,Y 565.495,Z 1080.009,A -85,B 0,C 180,E1 26527.105,E2 26527.105} C_VEL
LIN {X 0,Y 567.286,Z 1065.414,A -85,B 0,C 180,E1 26525.194,E2 26525.194} C_VEL
LIN {X 0,Y 569.521,Z 1048.514,A -85,B 0,C 180,E1 26523.235,E2 26523.235} C_VEL
LIN {X 0,Y 571.832,Z 1031.045,A -85,B 0,C 180,E1 26521.487,E2 26521.487} C_VEL
LIN {X 0,Y 574.24,Z 1013.168,A -85,B 0,C 180,E1 26519.902,E2 26519.902} C_VEL
LIN {X 0,Y 576.948,Z 992.409,A -85,B 0,C 180,E1 26518.314,E2 26518.314} C_VEL
LIN {X 0,Y 579.449,Z 972.858,A -85,B 0,C 180,E1 26517.014,E2 26517.014} C_VEL
LIN {X 0,Y 582.148,Z 949.79,A -85,B 0,C 180,E1 26515.707,E2 26515.707} C_VEL
LIN {X 0,Y 584.257,Z 930.482,A -85,B 0,C 180,E1 26514.778,E2 26514.778} C_VEL
LIN {X 0,Y 586.595,Z 906.184,A -85,B 0,C 180,E1 26513.798,E2 26513.798} C_VEL
LIN {X 0,Y 588.437,Z 883.866,A -85,B 0,C 180,E1 26513.081,E2 26513.081} C_VEL
LIN {X 0,Y 590.189,Z 859.121,A -85,B 0,C 180,E1 26512.464,E2 26512.464} C_VEL
LIN {X 0,Y 591.262,Z 835.898,A -85,B 0,C 180,E1 26512.051,E2 26512.051} C_VEL
LIN {X 0,Y 596.556,Z 601.976,A -85,B 0,C 180,E1 26508.902,E2 26508.902} C_VEL
LIN {X 0,Y 598.903,Z 496.812,A -85,B 0,C 180,E1 26507.466,E2 26507.466} C_VEL
LIN {X 0,Y 597.244,Z 489.81,A -85,B 0,C 180,E1 26507.216,E2 26507.216} C_VEL
LIN {X 0,Y 582.148,Z 463.955,A -85,B 0,C 180,E1 26505.463,E2 26505.463} C_VEL
LIN {X 0,Y 571.814,Z 447.252,A -85,B 0,C 180,E1 26504.173,E2 26504.173} C_VEL
LIN {X 0,Y 564.395,Z 429.547,A -85,B 0,C 180,E1 26501.633,E2 26501.633} C_VEL
LIN {X 0,Y 561.435,Z 422.45,A -85,B 0,C 180,E1 26500.512,E2 26500.512} C_VEL
LIN {X 0,Y 561.44,Z 422.279,A -85,B 0,C 180,E1 26497.395,E2 26497.395} C_VEL
LIN {X 0,Y 561.413,Z 422.29,A -85,B 0,C 180,E1 26494.088,E2 26494.088} C_VEL
LIN {X 0,Y 561.447,Z 422.295,A -85,B 0,C 180,E1 26490.739,E2 26490.739} C_VEL
LIN {X 0,Y 561.441,Z 422.286,A -85,B 0,C 180,E1 26487.291,E2 26487.291} C_VEL
LIN {X 0,Y 561.42,Z 422.267,A -85,B 0,C 180,E1 26483.958,E2 26483.958} C_VEL
LIN {X 0,Y 561.432,Z 422.29,A -85,B 0,C 180,E1 26480.758,E2 26480.758} C_VEL
LIN {X 0,Y 561.437,Z 422.291,A -85,B 0,C 180,E1 26477.332,E2 26477.332} C_VEL
LIN {X 0,Y 561.429,Z 422.267,A -85,B 0,C 180,E1 26474.017,E2 26474.017} C_VEL
LIN {X 0,Y 561.422,Z 422.292,A -85,B 0,C 180,E1 26470.778,E2 26470.778} C_VEL
LIN {X 0,Y 561.443,Z 422.277,A -85,B 0,C 180,E1 26467.367,E2 26467.367} C_VEL
LIN {X 0,Y 561.436,Z 422.274,A -85,B 0,C 180,E1 26463.983,E2 26463.983} C_VEL
LIN {X 0,Y 561.412,Z 422.299,A -85,B 0,C 180,E1 26460.714,E2 26460.714} C_VEL
LIN {X 0,Y 561.436,Z 422.265,A -85,B 0,C 180,E1 26457.448,E2 26457.448} C_VEL
LIN {X 0,Y 561.416,Z 422.294,A -85,B 0,C 180,E1 26454.173,E2 26454.173} C_VEL
LIN {X 0,Y 561.407,Z 422.279,A -85,B 0,C 180,E1 26450.776,E2 26450.776} C_VEL
LIN {X 0,Y 561.442,Z 422.278,A -85,B 0,C 180,E1 26447.555,E2 26447.555} C_VEL
LIN {X 0,Y 561.394,Z 422.298,A -85,B 0,C 180,E1 26444.292,E2 26444.292} C_VEL
LIN {X 0,Y 561.421,Z 422.27,A -85,B 0,C 180,E1 26440.978,E2 26440.978} C_VEL
LIN {X 0,Y 561.405,Z 422.296,A -85,B 0,C 180,E1 26437.816,E2 26437.816} C_VEL
LIN {X 0,Y 561.385,Z 422.297,A -85,B 0,C 180,E1 26434.467,E2 26434.467} C_VEL
LIN {X 0,Y 561.444,Z 422.27,A -85,B 0,C 180,E1 26431.259,E2 26431.259} C_VEL
LIN {X 0,Y 561.372,Z 422.294,A -85,B 0,C 180,E1 26428.17,E2 26428.17} C_VEL
LIN {X 0,Y 561.429,Z 422.3,A -85,B 0,C 180,E1 26425.007,E2 26425.007} C_VEL
LIN {X 0,Y 561.367,Z 422.302,A -85,B 0,C 180,E1 26421.825,E2 26421.825} C_VEL
LIN {X 0,Y 561.37,Z 422.221,A -85,B 0,C 180,E1 26418.502,E2 26418.502} C_VEL
LIN {X 0,Y 561.374,Z 422.277,A -85,B 0,C 180,E1 26415.43,E2 26415.43} C_VEL
LIN {X 0,Y 561.388,Z 422.558,A -85,B 0,C 180,E1 26413.881,E2 26413.881} C_VEL
LIN {X 0,Y 561.89,Z 424.313,A -85,B 0,C 180,E1 26413.672,E2 26413.672} C_VEL
LIN {X 0,Y 563.933,Z 427.189,A -85,B 0,C 180,E1 26413.405,E2 26413.405} C_VEL
LIN {X 0,Y 565.215,Z 428.628,A -85,B 0,C 180,E1 26413.247,E2 26413.247} C_VEL
LIN {X 0,Y 567.885,Z 432.509,A -85,B 0,C 180,E1 26412.906,E2 26412.906} C_VEL
LIN {X 0,Y 579.395,Z 449.11,A -85,B 0,C 180,E1 26411.498,E2 26411.498} C_VEL
LIN {X 0,Y 589.752,Z 464.671,A -85,B 0,C 180,E1 26410.294,E2 26410.294} C_VEL
LIN {X 0,Y 599.208,Z 480.602,A -85,B 0,C 180,E1 26409.222,E2 26409.222} C_VEL
LIN {X 0,Y 594.357,Z 684.334,A -85,B 0,C 180,E1 26406.473,E2 26406.473} C_VEL
LIN {X 0,Y 593.383,Z 692.03,A -85,B 0,C 180,E1 26406.432,E2 26406.432} C_VEL
LIN {X 0,Y 588.032,Z 712.567,A -85,B 0,C 180,E1 26406.535,E2 26406.535} C_VEL
LIN {X 0,Y 587.31,Z 719.168,A -85,B 0,C 180,E1 26406.49,E2 26406.49} C_VEL
LIN {X 0,Y 585.06,Z 807.92,A -85,B 0,C 180,E1 26405.271,E2 26405.271} C_VEL
LIN {X 0,Y 583.759,Z 833.113,A -85,B 0,C 180,E1 26404.758,E2 26404.758} C_VEL
LIN {X 0,Y 582.299,Z 853.765,A -85,B 0,C 180,E1 26404.197,E2 26404.197} C_VEL
LIN {X 0,Y 580.346,Z 877.084,A -85,B 0,C 180,E1 26403.4,E2 26403.4} C_VEL
LIN {X 0,Y 578.152,Z 898.337,A -85,B 0,C 180,E1 26402.499,E2 26402.499} C_VEL
LIN {X 0,Y 575.906,Z 918.214,A -85,B 0,C 180,E1 26401.507,E2 26401.507} C_VEL
LIN {X 0,Y 573.145,Z 939.998,A -85,B 0,C 180,E1 26400.219,E2 26400.219} C_VEL
LIN {X 0,Y 570.68,Z 958.122,A -85,B 0,C 180,E1 26398.977,E2 26398.977} C_VEL
LIN {X 0,Y 567.711,Z 979.151,A -85,B 0,C 180,E1 26397.311,E2 26397.311} C_VEL
LIN {X 0,Y 565.259,Z 995.741,A -85,B 0,C 180,E1 26395.792,E2 26395.792} C_VEL
LIN {X 0,Y 562.717,Z 1012.97,A -85,B 0,C 180,E1 26394.011,E2 26394.011} C_VEL
LIN {X 0,Y 560.377,Z 1028.744,A -85,B 0,C 180,E1 26392.117,E2 26392.117} C_VEL
LIN {X 0,Y 558.306,Z 1043.487,A -85,B 0,C 180,E1 26390.112,E2 26390.112} C_VEL
LIN {X 0,Y 556.432,Z 1057.526,A -85,B 0,C 180,E1 26387.896,E2 26387.896} C_VEL
LIN {X 0,Y 555.019,Z 1069.177,A -85,B 0,C 180,E1 26385.785,E2 26385.785} C_VEL
LIN {X 0,Y 553.794,Z 1080.874,A -85,B 0,C 180,E1 26383.299,E2 26383.299} C_VEL
LIN {X 0,Y 553.054,Z 1089.419,A -85,B 0,C 180,E1 26381.154,E2 26381.154} C_VEL
LIN {X 0,Y 552.445,Z 1098.071,A -85,B 0,C 180,E1 26378.535,E2 26378.535} C_VEL
LIN {X 0,Y 552.155,Z 1103.842,A -85,B 0,C 180,E1 26376.342,E2 26376.342} C_VEL
LIN {X 0,Y 551.983,Z 1109.006,A -85,B 0,C 180,E1 26373.843,E2 26373.843} C_VEL
LIN {X 0,Y 551.919,Z 1112.29,A -85,B 0,C 180,E1 26371.453,E2 26371.453} C_VEL
LIN {X 0,Y 551.917,Z 1114.064,A -85,B 0,C 180,E1 26369.377,E2 26369.377} C_VEL
LIN {X 0,Y 551.908,Z 1114.866,A -85,B 0,C 180,E1 26366.884,E2 26366.884} C_VEL
LIN {X 0,Y 551.914,Z 1114.04,A -85,B 0,C 180,E1 26364.49,E2 26364.49} C_VEL
LIN {X 0,Y 551.939,Z 1112.114,A -85,B 0,C 180,E1 26362.285,E2 26362.285} C_VEL
LIN {X 0,Y 552.018,Z 1108.112,A -85,B 0,C 180,E1 26359.597,E2 26359.597} C_VEL
LIN {X 0,Y 552.178,Z 1103.321,A -85,B 0,C 180,E1 26357.343,E2 26357.343} C_VEL
LIN {X 0,Y 552.565,Z 1096.355,A -85,B 0,C 180,E1 26354.788,E2 26354.788} C_VEL
LIN {X 0,Y 553.15,Z 1088.222,A -85,B 0,C 180,E1 26352.43,E2 26352.43} C_VEL
LIN {X 0,Y 554.057,Z 1078.545,A -85,B 0,C 180,E1 26350.057,E2 26350.057} C_VEL
LIN {X 0,Y 555.236,Z 1067.313,A -85,B 0,C 180,E1 26347.764,E2 26347.764} C_VEL
LIN {X 0,Y 556.767,Z 1055.024,A -85,B 0,C 180,E1 26345.577,E2 26345.577} C_VEL
LIN {X 0,Y 558.672,Z 1040.875,A -85,B 0,C 180,E1 26343.42,E2 26343.42} C_VEL
LIN {X 0,Y 560.684,Z 1026.908,A -85,B 0,C 180,E1 26341.545,E2 26341.545} C_VEL
LIN {X 0,Y 563.308,Z 1009.364,A -85,B 0,C 180,E1 26339.492,E2 26339.492} C_VEL
LIN {X 0,Y 565.73,Z 993.408,A -85,B 0,C 180,E1 26337.859,E2 26337.859} C_VEL
LIN {X 0,Y 568.698,Z 973.598,A -85,B 0,C 180,E1 26336.086,E2 26336.086} C_VEL
LIN {X 0,Y 571.375,Z 955.172,A -85,B 0,C 180,E1 26334.664,E2 26334.664} C_VEL
LIN {X 0,Y 574.291,Z 934.396,A -85,B 0,C 180,E1 26333.268,E2 26333.268} C_VEL
LIN {X 0,Y 576.888,Z 913.541,A -85,B 0,C 180,E1 26332.082,E2 26332.082} C_VEL
LIN {X 0,Y 579.309,Z 892.884,A -85,B 0,C 180,E1 26331.077,E2 26331.077} C_VEL
LIN {X 0,Y 581.599,Z 869.6,A -85,B 0,C 180,E1 26330.146,E2 26330.146} C_VEL
LIN {X 0,Y 583.416,Z 848.105,A -85,B 0,C 180,E1 26329.448,E2 26329.448} C_VEL
LIN {X 0,Y 585.137,Z 822.515,A -85,B 0,C 180,E1 26328.816,E2 26328.816} C_VEL
LIN {X 0,Y 586.126,Z 800.681,A -85,B 0,C 180,E1 26328.426,E2 26328.426} C_VEL
LIN {X 0,Y 592.728,Z 550.426,A -85,B 0,C 180,E1 26324.987,E2 26324.987} C_VEL
LIN {X 0,Y 594.487,Z 483.75,A -85,B 0,C 180,E1 26324.054,E2 26324.054} C_VEL
LIN {X 0,Y 583.809,Z 466.359,A -85,B 0,C 180,E1 26322.722,E2 26322.722} C_VEL
LIN {X 0,Y 571.385,Z 448.664,A -85,B 0,C 180,E1 26321.113,E2 26321.113} C_VEL
LIN {X 0,Y 564.075,Z 438.72,A -85,B 0,C 180,E1 26320.117,E2 26320.117} C_VEL
LIN {X 0,Y 560.543,Z 433.996,A -85,B 0,C 180,E1 26319.621,E2 26319.621} C_VEL
LIN {X 0,Y 557.78,Z 430.242,A -85,B 0,C 180,E1 26319.224,E2 26319.224} C_VEL
LIN {X 0,Y 556.774,Z 428.809,A -85,B 0,C 180,E1 26319.076,E2 26319.076} C_VEL
LIN {X 0,Y 554.293,Z 425.945,A -85,B 0,C 180,E1 26318.719,E2 26318.719} C_VEL
LIN {X 0,Y 553.583,Z 424.036,A -85,B 0,C 180,E1 26318.546,E2 26318.546} C_VEL
LIN {X 0,Y 553.433,Z 423.302,A -85,B 0,C 180,E1 26318.294,E2 26318.294} C_VEL
LIN {X 0,Y 553.458,Z 423.219,A -85,B 0,C 180,E1 26315.192,E2 26315.192} C_VEL
LIN {X 0,Y 553.429,Z 423.26,A -85,B 0,C 180,E1 26311.963,E2 26311.963} C_VEL
LIN {X 0,Y 553.502,Z 423.205,A -85,B 0,C 180,E1 26308.819,E2 26308.819} C_VEL
LIN {X 0,Y 553.443,Z 423.291,A -85,B 0,C 180,E1 26305.582,E2 26305.582} C_VEL
LIN {X 0,Y 553.474,Z 423.288,A -85,B 0,C 180,E1 26302.295,E2 26302.295} C_VEL
LIN {X 0,Y 553.474,Z 423.273,A -85,B 0,C 180,E1 26299.086,E2 26299.086} C_VEL
LIN {X 0,Y 553.45,Z 423.263,A -85,B 0,C 180,E1 26295.724,E2 26295.724} C_VEL
LIN {X 0,Y 553.505,Z 423.27,A -85,B 0,C 180,E1 26292.52,E2 26292.52} C_VEL
LIN {X 0,Y 553.466,Z 423.287,A -85,B 0,C 180,E1 26289.253,E2 26289.253} C_VEL
LIN {X 0,Y 553.474,Z 423.272,A -85,B 0,C 180,E1 26285.806,E2 26285.806} C_VEL
LIN {X 0,Y 553.498,Z 423.257,A -85,B 0,C 180,E1 26282.485,E2 26282.485} C_VEL
LIN {X 0,Y 553.475,Z 423.285,A -85,B 0,C 180,E1 26279.172,E2 26279.172} C_VEL
LIN {X 0,Y 553.489,Z 423.276,A -85,B 0,C 180,E1 26275.716,E2 26275.716} C_VEL
LIN {X 0,Y 553.498,Z 423.257,A -85,B 0,C 180,E1 26272.422,E2 26272.422} C_VEL
LIN {X 0,Y 553.483,Z 423.276,A -85,B 0,C 180,E1 26269.065,E2 26269.065} C_VEL
LIN {X 0,Y 553.508,Z 423.282,A -85,B 0,C 180,E1 26265.671,E2 26265.671} C_VEL
LIN {X 0,Y 553.49,Z 423.271,A -85,B 0,C 180,E1 26262.224,E2 26262.224} C_VEL
LIN {X 0,Y 553.489,Z 423.252,A -85,B 0,C 180,E1 26258.931,E2 26258.931} C_VEL
LIN {X 0,Y 553.499,Z 423.284,A -85,B 0,C 180,E1 26255.563,E2 26255.563} C_VEL
LIN {X 0,Y 553.484,Z 423.263,A -85,B 0,C 180,E1 26252.102,E2 26252.102} C_VEL
LIN {X 0,Y 553.496,Z 423.255,A -85,B 0,C 180,E1 26248.891,E2 26248.891} C_VEL
LIN {X 0,Y 553.48,Z 423.271,A -85,B 0,C 180,E1 26245.566,E2 26245.566} C_VEL
LIN {X 0,Y 553.477,Z 423.278,A -85,B 0,C 180,E1 26242.104,E2 26242.104} C_VEL
LIN {X 0,Y 553.554,Z 423.592,A -85,B 0,C 180,E1 26241.069,E2 26241.069} C_VEL
LIN {X 0,Y 560.725,Z 439.858,A -85,B 0,C 180,E1 26238.307,E2 26238.307} C_VEL
LIN {X 0,Y 563.914,Z 446.926,A -85,B 0,C 180,E1 26237.226,E2 26237.226} C_VEL
LIN {X 0,Y 576.981,Z 467.074,A -85,B 0,C 180,E1 26235.424,E2 26235.424} C_VEL
LIN {X 0,Y 589.539,Z 487.931,A -85,B 0,C 180,E1 26233.807,E2 26233.807} C_VEL
LIN {X 0,Y 593.755,Z 495.882,A -85,B 0,C 180,E1 26233.276,E2 26233.276} C_VEL
LIN {X 0,Y 594.429,Z 500.666,A -85,B 0,C 180,E1 26233.134,E2 26233.134} C_VEL
LIN {X 0,Y 588.237,Z 734.829,A -85,B 0,C 180,E1 26229.909,E2 26229.909} C_VEL
LIN {X 0,Y 585.469,Z 840.192,A -85,B 0,C 180,E1 26228.451,E2 26228.451} C_VEL
LIN {X 0,Y 583.903,Z 866.292,A -85,B 0,C 180,E1 26227.931,E2 26227.931} C_VEL
LIN {X 0,Y 582.186,Z 888.113,A -85,B 0,C 180,E1 26227.341,E2 26227.341} C_VEL
LIN {X 0,Y 579.929,Z 912.367,A -85,B 0,C 180,E1 26226.501,E2 26226.501} C_VEL
LIN {X 0,Y 577.69,Z 933,A -85,B 0,C 180,E1 26225.622,E2 26225.622} C_VEL
LIN {X 0,Y 575.031,Z 955.443,A -85,B 0,C 180,E1 26224.491,E2 26224.491} C_VEL
LIN {X 0,Y 572.229,Z 976.592,A -85,B 0,C 180,E1 26223.216,E2 26223.216} C_VEL
LIN {X 0,Y 569.417,Z 997.171,A -85,B 0,C 180,E1 26221.789,E2 26221.789} C_VEL
LIN {X 0,Y 566.594,Z 1016.785,A -85,B 0,C 180,E1 26220.196,E2 26220.196} C_VEL
LIN {X 0,Y 564.041,Z 1034.678,A -85,B 0,C 180,E1 26218.546,E2 26218.546} C_VEL
LIN {X 0,Y 561.418,Z 1052.919,A -85,B 0,C 180,E1 26216.611,E2 26216.611} C_VEL
LIN {X 0,Y 559.313,Z 1068.373,A -85,B 0,C 180,E1 26214.747,E2 26214.747} C_VEL
LIN {X 0,Y 557.184,Z 1084.805,A -85,B 0,C 180,E1 26212.472,E2 26212.472} C_VEL
LIN {X 0,Y 555.752,Z 1097.008,A -85,B 0,C 180,E1 26210.539,E2 26210.539} C_VEL
LIN {X 0,Y 554.342,Z 1110.507,A -85,B 0,C 180,E1 26208.074,E2 26208.074} C_VEL
LIN {X 0,Y 553.439,Z 1120.489,A -85,B 0,C 180,E1 26205.939,E2 26205.939} C_VEL
LIN {X 0,Y 552.733,Z 1130.26,A -85,B 0,C 180,E1 26203.495,E2 26203.495} C_VEL
LIN {X 0,Y 552.297,Z 1137.803,A -85,B 0,C 180,E1 26201.17,E2 26201.17} C_VEL
LIN {X 0,Y 552.058,Z 1143.931,A -85,B 0,C 180,E1 26198.856,E2 26198.856} C_VEL
LIN {X 0,Y 551.954,Z 1148.869,A -85,B 0,C 180,E1 26196.344,E2 26196.344} C_VEL
LIN {X 0,Y 551.924,Z 1151.838,A -85,B 0,C 180,E1 26194.156,E2 26194.156} C_VEL
LIN {X 0,Y 551.904,Z 1153.791,A -85,B 0,C 180,E1 26191.661,E2 26191.661} C_VEL
LIN {X 0,Y 551.89,Z 1154.026,A -85,B 0,C 180,E1 26189.377,E2 26189.377} C_VEL
LIN {X 0,Y 551.893,Z 1153.128,A -85,B 0,C 180,E1 26187.3,E2 26187.3} C_VEL
LIN {X 0,Y 551.91,Z 1150.908,A -85,B 0,C 180,E1 26185.011,E2 26185.011} C_VEL
LIN {X 0,Y 551.973,Z 1146.802,A -85,B 0,C 180,E1 26182.506,E2 26182.506} C_VEL
LIN {X 0,Y 552.135,Z 1142.122,A -85,B 0,C 180,E1 26180.409,E2 26180.409} C_VEL
LIN {X 0,Y 552.439,Z 1135.319,A -85,B 0,C 180,E1 26177.986,E2 26177.986} C_VEL
LIN {X 0,Y 552.937,Z 1127.046,A -85,B 0,C 180,E1 26175.656,E2 26175.656} C_VEL
LIN {X 0,Y 553.633,Z 1118.181,A -85,B 0,C 180,E1 26173.528,E2 26173.528} C_VEL
LIN {X 0,Y 554.771,Z 1106.103,A -85,B 0,C 180,E1 26171.069,E2 26171.069} C_VEL
LIN {X 0,Y 556.053,Z 1094.474,A -85,B 0,C 180,E1 26169.032,E2 26169.032} C_VEL
LIN {X 0,Y 557.856,Z 1079.734,A -85,B 0,C 180,E1 26166.776,E2 26166.776} C_VEL
LIN {X 0,Y 559.748,Z 1065.136,A -85,B 0,C 180,E1 26164.84,E2 26164.84} C_VEL
LIN {X 0,Y 562.121,Z 1048.177,A -85,B 0,C 180,E1 26162.854,E2 26162.854} C_VEL
LIN {X 0,Y 564.544,Z 1030.672,A -85,B 0,C 180,E1 26161.084,E2 26161.084} C_VEL
LIN {X 0,Y 567.168,Z 1012.15,A -85,B 0,C 180,E1 26159.428,E2 26159.428} C_VEL
LIN {X 0,Y 569.92,Z 992.089,A -85,B 0,C 180,E1 26157.887,E2 26157.887} C_VEL
LIN {X 0,Y 572.475,Z 972.984,A -85,B 0,C 180,E1 26156.604,E2 26156.604} C_VEL
LIN {X 0,Y 575.255,Z 950.341,A -85,B 0,C 180,E1 26155.301,E2 26155.301} C_VEL
LIN {X 0,Y 577.583,Z 929.917,A -85,B 0,C 180,E1 26154.31,E2 26154.31} C_VEL
LIN {X 0,Y 580.038,Z 905.521,A -85,B 0,C 180,E1 26153.322,E2 26153.322} C_VEL
LIN {X 0,Y 581.933,Z 883.57,A -85,B 0,C 180,E1 26152.614,E2 26152.614} C_VEL
LIN {X 0,Y 583.75,Z 858.862,A -85,B 0,C 180,E1 26151.994,E2 26151.994} C_VEL
LIN {X 0,Y 584.866,Z 835.564,A -85,B 0,C 180,E1 26151.576,E2 26151.576} C_VEL
LIN {X 0,Y 590.422,Z 601.793,A -85,B 0,C 180,E1 26148.401,E2 26148.401} C_VEL
LIN {X 0,Y 592.864,Z 498.603,A -85,B 0,C 180,E1 26146.98,E2 26146.98} C_VEL
LIN {X 0,Y 591.676,Z 493.896,A -85,B 0,C 180,E1 26146.802,E2 26146.802} C_VEL
LIN {X 0,Y 577.243,Z 469.095,A -85,B 0,C 180,E1 26145.093,E2 26145.093} C_VEL
LIN {X 0,Y 563.557,Z 447.296,A -85,B 0,C 180,E1 26143.365,E2 26143.365} C_VEL
LIN {X 0,Y 558.209,Z 434.482,A -85,B 0,C 180,E1 26141.511,E2 26141.511} C_VEL
LIN {X 0,Y 553.518,Z 423.488,A -85,B 0,C 180,E1 26139.753,E2 26139.753} C_VEL
LIN {X 0,Y 553.473,Z 423.266,A -85,B 0,C 180,E1 26136.339,E2 26136.339} C_VEL
LIN {X 0,Y 553.499,Z 423.26,A -85,B 0,C 180,E1 26133.048,E2 26133.048} C_VEL
LIN {X 0,Y 553.489,Z 423.266,A -85,B 0,C 180,E1 26129.664,E2 26129.664} C_VEL
LIN {X 0,Y 553.489,Z 423.285,A -85,B 0,C 180,E1 26126.27,E2 26126.27} C_VEL
LIN {X 0,Y 553.494,Z 423.268,A -85,B 0,C 180,E1 26122.88,E2 26122.88} C_VEL
LIN {X 0,Y 553.495,Z 423.259,A -85,B 0,C 180,E1 26119.524,E2 26119.524} C_VEL
LIN {X 0,Y 553.496,Z 423.283,A -85,B 0,C 180,E1 26116.153,E2 26116.153} C_VEL
LIN {X 0,Y 553.484,Z 423.27,A -85,B 0,C 180,E1 26112.839,E2 26112.839} C_VEL
LIN {X 0,Y 553.495,Z 423.259,A -85,B 0,C 180,E1 26109.462,E2 26109.462} C_VEL
LIN {X 0,Y 553.505,Z 423.281,A -85,B 0,C 180,E1 26106.014,E2 26106.014} C_VEL
LIN {X 0,Y 553.471,Z 423.259,A -85,B 0,C 180,E1 26102.692,E2 26102.692} C_VEL
LIN {X 0,Y 553.503,Z 423.277,A -85,B 0,C 180,E1 26099.379,E2 26099.379} C_VEL
LIN {X 0,Y 553.493,Z 423.272,A -85,B 0,C 180,E1 26095.96,E2 26095.96} C_VEL
LIN {X 0,Y 553.463,Z 423.262,A -85,B 0,C 180,E1 26092.63,E2 26092.63} C_VEL
LIN {X 0,Y 553.502,Z 423.285,A -85,B 0,C 180,E1 26089.277,E2 26089.277} C_VEL
LIN {X 0,Y 553.47,Z 423.256,A -85,B 0,C 180,E1 26085.964,E2 26085.964} C_VEL
LIN {X 0,Y 553.461,Z 423.279,A -85,B 0,C 180,E1 26082.657,E2 26082.657} C_VEL
LIN {X 0,Y 553.509,Z 423.273,A -85,B 0,C 180,E1 26079.35,E2 26079.35} C_VEL
LIN {X 0,Y 553.442,Z 423.259,A -85,B 0,C 180,E1 26076.241,E2 26076.241} C_VEL
LIN {X 0,Y 553.482,Z 423.278,A -85,B 0,C 180,E1 26072.919,E2 26072.919} C_VEL
LIN {X 0,Y 553.445,Z 423.286,A -85,B 0,C 180,E1 26069.851,E2 26069.851} C_VEL
LIN {X 0,Y 553.437,Z 423.274,A -85,B 0,C 180,E1 26066.397,E2 26066.397} C_VEL
LIN {X 0,Y 553.489,Z 423.264,A -85,B 0,C 180,E1 26063.147,E2 26063.147} C_VEL
LIN {X 0,Y 553.417,Z 423.258,A -85,B 0,C 180,E1 26060.104,E2 26060.104} C_VEL
LIN {X 0,Y 553.473,Z 423.205,A -85,B 0,C 180,E1 26056.93,E2 26056.93} C_VEL
LIN {X 0,Y 553.492,Z 423.491,A -85,B 0,C 180,E1 26054.718,E2 26054.718} C_VEL
LIN {X 0,Y 553.895,Z 425.115,A -85,B 0,C 180,E1 26054.516,E2 26054.516} C_VEL
LIN {X 0,Y 555.859,Z 428.094,A -85,B 0,C 180,E1 26054.243,E2 26054.243} C_VEL
LIN {X 0,Y 557.281,Z 429.652,A -85,B 0,C 180,E1 26054.062,E2 26054.062} C_VEL
LIN {X 0,Y 560.069,Z 433.628,A -85,B 0,C 180,E1 26053.693,E2 26053.693} C_VEL
LIN {X 0,Y 573.996,Z 453.378,A -85,B 0,C 180,E1 26051.941,E2 26051.941} C_VEL
LIN {X 0,Y 586.301,Z 472.144,A -85,B 0,C 180,E1 26050.481,E2 26050.481} C_VEL
LIN {X 0,Y 593.128,Z 483.874,A -85,B 0,C 180,E1 26049.69,E2 26049.69} C_VEL
LIN {X 0,Y 587.31,Z 719.168,A -85,B 0,C 180,E1 26046.49,E2 26046.49} C_VEL
LIN {X 0,Y 586.363,Z 726.862,A -85,B 0,C 180,E1 26046.446,E2 26046.446} C_VEL
LIN {X 0,Y 580.954,Z 747.388,A -85,B 0,C 180,E1 26046.555,E2 26046.555} C_VEL
LIN {X 0,Y 580.203,Z 753.992,A -85,B 0,C 180,E1 26046.512,E2 26046.512} C_VEL
LIN {X 0,Y 578.66,Z 810.211,A -85,B 0,C 180,E1 26045.719,E2 26045.719} C_VEL
LIN {X 0,Y 577.311,Z 834.219,A -85,B 0,C 180,E1 26045.214,E2 26045.214} C_VEL
LIN {X 0,Y 575.785,Z 854.931,A -85,B 0,C 180,E1 26044.643,E2 26044.643} C_VEL
LIN {X 0,Y 573.606,Z 879.369,A -85,B 0,C 180,E1 26043.785,E2 26043.785} C_VEL
LIN {X 0,Y 571.417,Z 899.69,A -85,B 0,C 180,E1 26042.908,E2 26042.908} C_VEL
LIN {X 0,Y 568.903,Z 921.052,A -85,B 0,C 180,E1 26041.822,E2 26041.822} C_VEL
LIN {X 0,Y 565.997,Z 942.546,A -85,B 0,C 180,E1 26040.51,E2 26040.51} C_VEL
LIN {X 0,Y 563.098,Z 963.164,A -85,B 0,C 180,E1 26039.055,E2 26039.055} C_VEL
LIN {X 0,Y 560.24,Z 981.964,A -85,B 0,C 180,E1 26037.498,E2 26037.498} C_VEL
LIN {X 0,Y 557.606,Z 999.074,A -85,B 0,C 180,E1 26035.89,E2 26035.89} C_VEL
LIN {X 0,Y 554.764,Z 1017.192,A -85,B 0,C 180,E1 26033.925,E2 26033.925} C_VEL
LIN {X 0,Y 552.5,Z 1031.985,A -85,B 0,C 180,E1 26032.089,E2 26032.089} C_VEL
LIN {X 0,Y 550.103,Z 1048.251,A -85,B 0,C 180,E1 26029.76,E2 26029.76} C_VEL
LIN {X 0,Y 548.406,Z 1060.545,A -85,B 0,C 180,E1 26027.727,E2 26027.727} C_VEL
LIN {X 0,Y 546.752,Z 1073.869,A -85,B 0,C 180,E1 26025.16,E2 26025.16} C_VEL
LIN {X 0,Y 545.743,Z 1083.311,A -85,B 0,C 180,E1 26023.024,E2 26023.024} C_VEL
LIN {X 0,Y 544.875,Z 1093.204,A -85,B 0,C 180,E1 26020.36,E2 26020.36} C_VEL
LIN {X 0,Y 544.407,Z 1099.974,A -85,B 0,C 180,E1 26018.124,E2 26018.124} C_VEL
LIN {X 0,Y 544.102,Z 1106.169,A -85,B 0,C 180,E1 26015.589,E2 26015.589} C_VEL
LIN {X 0,Y 543.96,Z 1110.447,A -85,B 0,C 180,E1 26013.161,E2 26013.161} C_VEL
LIN {X 0,Y 543.91,Z 1113.065,A -85,B 0,C 180,E1 26011.053,E2 26011.053} C_VEL
LIN {X 0,Y 543.895,Z 1114.835,A -85,B 0,C 180,E1 26008.525,E2 26008.525} C_VEL
LIN {X 0,Y 543.905,Z 1115.007,A -85,B 0,C 180,E1 26006.205,E2 26006.205} C_VEL
LIN {X 0,Y 543.93,Z 1113.965,A -85,B 0,C 180,E1 26003.879,E2 26003.879} C_VEL
LIN {X 0,Y 543.968,Z 1111.158,A -85,B 0,C 180,E1 26001.224,E2 26001.224} C_VEL
LIN {X 0,Y 544.055,Z 1107.436,A -85,B 0,C 180,E1 25998.981,E2 25998.981} C_VEL
LIN {X 0,Y 544.31,Z 1101.701,A -85,B 0,C 180,E1 25996.4,E2 25996.4} C_VEL
LIN {X 0,Y 544.741,Z 1094.745,A -85,B 0,C 180,E1 25994.018,E2 25994.018} C_VEL
LIN {X 0,Y 545.42,Z 1086.73,A -85,B 0,C 180,E1 25991.73,E2 25991.73} C_VEL
LIN {X 0,Y 546.498,Z 1076.101,A -85,B 0,C 180,E1 25989.22,E2 25989.22} C_VEL
LIN {X 0,Y 547.758,Z 1065.716,A -85,B 0,C 180,E1 25987.119,E2 25987.119} C_VEL
LIN {X 0,Y 549.636,Z 1051.761,A -85,B 0,C 180,E1 25984.69,E2 25984.69} C_VEL
LIN {X 0,Y 551.605,Z 1038.216,A -85,B 0,C 180,E1 25982.651,E2 25982.651} C_VEL
LIN {X 0,Y 554.312,Z 1020.795,A -85,B 0,C 180,E1 25980.379,E2 25980.379} C_VEL
LIN {X 0,Y 556.683,Z 1005.82,A -85,B 0,C 180,E1 25978.677,E2 25978.677} C_VEL
LIN {X 0,Y 559.711,Z 986.993,A -85,B 0,C 180,E1 25976.801,E2 25976.801} C_VEL
LIN {X 0,Y 562.491,Z 969.212,A -85,B 0,C 180,E1 25975.269,E2 25975.269} C_VEL
LIN {X 0,Y 565.584,Z 948.93,A -85,B 0,C 180,E1 25973.74,E2 25973.74} C_VEL
LIN {X 0,Y 568.392,Z 928.688,A -85,B 0,C 180,E1 25972.443,E2 25972.443} C_VEL
LIN {X 0,Y 571.196,Z 907.247,A -85,B 0,C 180,E1 25971.258,E2 25971.258} C_VEL
LIN {X 0,Y 573.763,Z 884.868,A -85,B 0,C 180,E1 25970.24,E2 25970.24} C_VEL
LIN {X 0,Y 575.79,Z 864.534,A -85,B 0,C 180,E1 25969.465,E2 25969.465} C_VEL
LIN {X 0,Y 577.853,Z 839.707,A -85,B 0,C 180,E1 25968.715,E2 25968.715} C_VEL
LIN {X 0,Y 579.171,Z 819.034,A -85,B 0,C 180,E1 25968.24,E2 25968.24} C_VEL
LIN {X 0,Y 580.237,Z 793.917,A -85,B 0,C 180,E1 25967.817,E2 25967.817} C_VEL
LIN {X 0,Y 587.121,Z 543.54,A -85,B 0,C 180,E1 25964.353,E2 25964.353} C_VEL
LIN {X 0,Y 588.641,Z 487.091,A -85,B 0,C 180,E1 25963.552,E2 25963.552} C_VEL
LIN {X 0,Y 578.614,Z 470.846,A -85,B 0,C 180,E1 25962.273,E2 25962.273} C_VEL
LIN {X 0,Y 566.825,Z 454.07,A -85,B 0,C 180,E1 25960.711,E2 25960.711} C_VEL
LIN {X 0,Y 559.431,Z 444.01,A -85,B 0,C 180,E1 25959.682,E2 25959.682} C_VEL
LIN {X 0,Y 556.366,Z 439.939,A -85,B 0,C 180,E1 25959.243,E2 25959.243} C_VEL
LIN {X 0,Y 552.774,Z 435.048,A -85,B 0,C 180,E1 25958.713,E2 25958.713} C_VEL
LIN {X 0,Y 549.932,Z 431.181,A -85,B 0,C 180,E1 25958.284,E2 25958.284} C_VEL
LIN {X 0,Y 548.938,Z 429.887,A -85,B 0,C 180,E1 25958.133,E2 25958.133} C_VEL
LIN {X 0,Y 546.425,Z 427.128,A -85,B 0,C 180,E1 25957.758,E2 25957.758} C_VEL
LIN {X 0,Y 545.623,Z 425,A -85,B 0,C 180,E1 25957.56,E2 25957.56} C_VEL
LIN {X 0,Y 545.519,Z 424.243,A -85,B 0,C 180,E1 25957.219,E2 25957.219} C_VEL
LIN {X 0,Y 545.487,Z 424.248,A -85,B 0,C 180,E1 25953.992,E2 25953.992} C_VEL
LIN {X 0,Y 545.559,Z 424.195,A -85,B 0,C 180,E1 25950.754,E2 25950.754} C_VEL
LIN {X 0,Y 545.495,Z 424.235,A -85,B 0,C 180,E1 25947.629,E2 25947.629} C_VEL
LIN {X 0,Y 545.535,Z 424.254,A -85,B 0,C 180,E1 25944.355,E2 25944.355} C_VEL
LIN {X 0,Y 545.519,Z 424.268,A -85,B 0,C 180,E1 25941.28,E2 25941.28} C_VEL
LIN {X 0,Y 545.517,Z 424.278,A -85,B 0,C 180,E1 25937.824,E2 25937.824} C_VEL
LIN {X 0,Y 545.572,Z 424.261,A -85,B 0,C 180,E1 25934.542,E2 25934.542} C_VEL
LIN {X 0,Y 545.526,Z 424.252,A -85,B 0,C 180,E1 25931.203,E2 25931.203} C_VEL
LIN {X 0,Y 545.53,Z 424.263,A -85,B 0,C 180,E1 25927.795,E2 25927.795} C_VEL
LIN {X 0,Y 545.564,Z 424.275,A -85,B 0,C 180,E1 25924.52,E2 25924.52} C_VEL
LIN {X 0,Y 545.532,Z 424.251,A -85,B 0,C 180,E1 25921.155,E2 25921.155} C_VEL
LIN {X 0,Y 545.548,Z 424.248,A -85,B 0,C 180,E1 25917.794,E2 25917.794} C_VEL
LIN {X 0,Y 545.56,Z 424.266,A -85,B 0,C 180,E1 25914.386,E2 25914.386} C_VEL
LIN {X 0,Y 545.544,Z 424.263,A -85,B 0,C 180,E1 25911.037,E2 25911.037} C_VEL
LIN {X 0,Y 545.556,Z 424.245,A -85,B 0,C 180,E1 25907.617,E2 25907.617} C_VEL
LIN {X 0,Y 545.552,Z 424.259,A -85,B 0,C 180,E1 25904.261,E2 25904.261} C_VEL
LIN {X 0,Y 545.556,Z 424.277,A -85,B 0,C 180,E1 25900.848,E2 25900.848} C_VEL
LIN {X 0,Y 545.561,Z 424.243,A -85,B 0,C 180,E1 25897.363,E2 25897.363} C_VEL
LIN {X 0,Y 545.542,Z 424.245,A -85,B 0,C 180,E1 25894.02,E2 25894.02} C_VEL
LIN {X 0,Y 545.567,Z 424.272,A -85,B 0,C 180,E1 25890.582,E2 25890.582} C_VEL
LIN {X 0,Y 545.564,Z 424.265,A -85,B 0,C 180,E1 25887.078,E2 25887.078} C_VEL
LIN {X 0,Y 545.534,Z 424.253,A -85,B 0,C 180,E1 25883.7,E2 25883.7} C_VEL
LIN {X 0,Y 545.568,Z 424.513,A -85,B 0,C 180,E1 25882.007,E2 25882.007} C_VEL
LIN {X 0,Y 547.152,Z 428.159,A -85,B 0,C 180,E1 25881.319,E2 25881.319} C_VEL
LIN {X 0,Y 553.431,Z 442.256,A -85,B 0,C 180,E1 25878.879,E2 25878.879} C_VEL
LIN {X 0,Y 555.371,Z 446.499,A -85,B 0,C 180,E1 25878.229,E2 25878.229} C_VEL
LIN {X 0,Y 565.753,Z 462.007,A -85,B 0,C 180,E1 25876.725,E2 25876.725} C_VEL
LIN {X 0,Y 578.813,Z 482.843,A -85,B 0,C 180,E1 25874.957,E2 25874.957} C_VEL
LIN {X 0,Y 588.327,Z 499.574,A -85,B 0,C 180,E1 25873.728,E2 25873.728} C_VEL
LIN {X 0,Y 588.611,Z 502.825,A -85,B 0,C 180,E1 25873.646,E2 25873.646} C_VEL
LIN {X 0,Y 582.157,Z 735.729,A -85,B 0,C 180,E1 25870.412,E2 25870.412} C_VEL
LIN {X 0,Y 579.284,Z 839.91,A -85,B 0,C 180,E1 25868.956,E2 25868.956} C_VEL
LIN {X 0,Y 577.651,Z 866.065,A -85,B 0,C 180,E1 25868.432,E2 25868.432} C_VEL
LIN {X 0,Y 575.844,Z 887.995,A -85,B 0,C 180,E1 25867.835,E2 25867.835} C_VEL
LIN {X 0,Y 573.454,Z 912.426,A -85,B 0,C 180,E1 25866.981,E2 25866.981} C_VEL
LIN {X 0,Y 571.118,Z 933.009,A -85,B 0,C 180,E1 25866.096,E2 25866.096} C_VEL
LIN {X 0,Y 568.327,Z 955.422,A -85,B 0,C 180,E1 25864.954,E2 25864.954} C_VEL
LIN {X 0,Y 565.526,Z 975.687,A -85,B 0,C 180,E1 25863.723,E2 25863.723} C_VEL
LIN {X 0,Y 562.763,Z 994.836,A -85,B 0,C 180,E1 25862.391,E2 25862.391} C_VEL
LIN {X 0,Y 559.657,Z 1015.396,A -85,B 0,C 180,E1 25860.729,E2 25860.729} C_VEL
LIN {X 0,Y 557.088,Z 1032.352,A -85,B 0,C 180,E1 25859.161,E2 25859.161} C_VEL
LIN {X 0,Y 554.231,Z 1051.292,A -85,B 0,C 180,E1 25857.158,E2 25857.158} C_VEL
LIN {X 0,Y 551.995,Z 1066.55,A -85,B 0,C 180,E1 25855.309,E2 25855.309} C_VEL
LIN {X 0,Y 549.82,Z 1082.382,A -85,B 0,C 180,E1 25853.13,E2 25853.13} C_VEL
LIN {X 0,Y 548.156,Z 1095.415,A -85,B 0,C 180,E1 25851.06,E2 25851.06} C_VEL
LIN {X 0,Y 546.717,Z 1108.092,A -85,B 0,C 180,E1 25848.777,E2 25848.777} C_VEL
LIN {X 0,Y 545.614,Z 1119.255,A -85,B 0,C 180,E1 25846.393,E2 25846.393} C_VEL
LIN {X 0,Y 544.881,Z 1128.384,A -85,B 0,C 180,E1 25844.127,E2 25844.127} C_VEL
LIN {X 0,Y 544.348,Z 1136.89,A -85,B 0,C 180,E1 25841.55,E2 25841.55} C_VEL
LIN {X 0,Y 544.113,Z 1142.602,A -85,B 0,C 180,E1 25839.413,E2 25839.413} C_VEL
LIN {X 0,Y 543.973,Z 1147.925,A -85,B 0,C 180,E1 25836.862,E2 25836.862} C_VEL
LIN {X 0,Y 543.93,Z 1151.319,A -85,B 0,C 180,E1 25834.428,E2 25834.428} C_VEL
LIN {X 0,Y 543.918,Z 1153.19,A -85,B 0,C 180,E1 25832.212,E2 25832.212} C_VEL
LIN {X 0,Y 543.898,Z 1153.787,A -85,B 0,C 180,E1 25829.579,E2 25829.579} C_VEL
LIN {X 0,Y 543.9,Z 1152.913,A -85,B 0,C 180,E1 25827.366,E2 25827.366} C_VEL
LIN {X 0,Y 543.916,Z 1150.823,A -85,B 0,C 180,E1 25825.119,E2 25825.119} C_VEL
LIN {X 0,Y 543.973,Z 1146.727,A -85,B 0,C 180,E1 25822.501,E2 25822.501} C_VEL
LIN {X 0,Y 544.145,Z 1141.835,A -85,B 0,C 180,E1 25820.267,E2 25820.267} C_VEL
LIN {X 0,Y 544.474,Z 1135.031,A -85,B 0,C 180,E1 25817.808,E2 25817.808} C_VEL
LIN {X 0,Y 545.041,Z 1126.344,A -85,B 0,C 180,E1 25815.335,E2 25815.335} C_VEL
LIN {X 0,Y 545.842,Z 1116.956,A -85,B 0,C 180,E1 25813.066,E2 25813.066} C_VEL
LIN {X 0,Y 547.028,Z 1105.229,A -85,B 0,C 180,E1 25810.68,E2 25810.68} C_VEL
LIN {X 0,Y 548.393,Z 1093.536,A -85,B 0,C 180,E1 25808.613,E2 25808.613} C_VEL
LIN {X 0,Y 550.433,Z 1077.86,A -85,B 0,C 180,E1 25806.217,E2 25806.217} C_VEL
LIN {X 0,Y 552.364,Z 1063.858,A -85,B 0,C 180,E1 25804.354,E2 25804.354} C_VEL
LIN {X 0,Y 555.018,Z 1045.743,A -85,B 0,C 180,E1 25802.244,E2 25802.244} C_VEL
LIN {X 0,Y 557.444,Z 1029.144,A -85,B 0,C 180,E1 25800.562,E2 25800.562} C_VEL
LIN {X 0,Y 560.339,Z 1009.778,A -85,B 0,C 180,E1 25798.836,E2 25798.836} C_VEL
LIN {X 0,Y 563.044,Z 990.881,A -85,B 0,C 180,E1 25797.386,E2 25797.386} C_VEL
LIN {X 0,Y 565.673,Z 972.053,A -85,B 0,C 180,E1 25796.116,E2 25796.116} C_VEL
LIN {X 0,Y 568.563,Z 949.366,A -85,B 0,C 180,E1 25794.807,E2 25794.807} C_VEL
LIN {X 0,Y 570.952,Z 929.33,A -85,B 0,C 180,E1 25793.83,E2 25793.83} C_VEL
LIN {X 0,Y 573.595,Z 904.105,A -85,B 0,C 180,E1 25792.811,E2 25792.811} C_VEL
LIN {X 0,Y 575.498,Z 882.919,A -85,B 0,C 180,E1 25792.127,E2 25792.127} C_VEL
LIN {X 0,Y 577.379,Z 858.041,A -85,B 0,C 180,E1 25791.503,E2 25791.503} C_VEL
LIN {X 0,Y 578.514,Z 835.076,A -85,B 0,C 180,E1 25791.089,E2 25791.089} C_VEL
LIN {X 0,Y 584.331,Z 601.74,A -85,B 0,C 180,E1 25787.891,E2 25787.891} C_VEL
LIN {X 0,Y 586.829,Z 500.216,A -85,B 0,C 180,E1 25786.478,E2 25786.478} C_VEL
LIN {X 0,Y 585.982,Z 497.647,A -85,B 0,C 180,E1 25786.362,E2 25786.362} C_VEL
LIN {X 0,Y 571.65,Z 473.105,A -85,B 0,C 180,E1 25784.628,E2 25784.628} C_VEL
LIN {X 0,Y 558.661,Z 452.327,A -85,B 0,C 180,E1 25782.959,E2 25782.959} C_VEL
LIN {X 0,Y 554.986,Z 446.417,A -85,B 0,C 180,E1 25782.433,E2 25782.433} C_VEL
LIN {X 0,Y 548.676,Z 431.783,A -85,B 0,C 180,E1 25780.175,E2 25780.175} C_VEL
LIN {X 0,Y 545.596,Z 424.453,A -85,B 0,C 180,E1 25778.941,E2 25778.941} C_VEL
LIN {X 0,Y 545.557,Z 424.263,A -85,B 0,C 180,E1 25775.535,E2 25775.535} C_VEL
LIN {X 0,Y 545.537,Z 424.257,A -85,B 0,C 180,E1 25772.136,E2 25772.136} C_VEL
LIN {X 0,Y 545.562,Z 424.243,A -85,B 0,C 180,E1 25768.818,E2 25768.818} C_VEL
LIN {X 0,Y 545.558,Z 424.257,A -85,B 0,C 180,E1 25765.369,E2 25765.369} C_VEL
LIN {X 0,Y 545.545,Z 424.272,A -85,B 0,C 180,E1 25761.956,E2 25761.956} C_VEL
LIN {X 0,Y 545.556,Z 424.248,A -85,B 0,C 180,E1 25758.597,E2 25758.597} C_VEL
LIN {X 0,Y 545.555,Z 424.254,A -85,B 0,C 180,E1 25755.194,E2 25755.194} C_VEL
LIN {X 0,Y 545.556,Z 424.27,A -85,B 0,C 180,E1 25751.842,E2 25751.842} C_VEL
LIN {X 0,Y 545.548,Z 424.241,A -85,B 0,C 180,E1 25748.431,E2 25748.431} C_VEL
LIN {X 0,Y 545.548,Z 424.266,A -85,B 0,C 180,E1 25745.047,E2 25745.047} C_VEL
LIN {X 0,Y 545.561,Z 424.257,A -85,B 0,C 180,E1 25741.68,E2 25741.68} C_VEL
LIN {X 0,Y 545.534,Z 424.253,A -85,B 0,C 180,E1 25738.425,E2 25738.425} C_VEL
LIN {X 0,Y 545.541,Z 424.278,A -85,B 0,C 180,E1 25734.953,E2 25734.953} C_VEL
LIN {X 0,Y 545.563,Z 424.238,A -85,B 0,C 180,E1 25731.675,E2 25731.675} C_VEL
LIN {X 0,Y 545.522,Z 424.273,A -85,B 0,C 180,E1 25728.368,E2 25728.368} C_VEL
LIN {X 0,Y 545.545,Z 424.257,A -85,B 0,C 180,E1 25724.996,E2 25724.996} C_VEL
LIN {X 0,Y 545.545,Z 424.25,A -85,B 0,C 180,E1 25721.697,E2 25721.697} C_VEL
LIN {X 0,Y 545.508,Z 424.277,A -85,B 0,C 180,E1 25718.381,E2 25718.381} C_VEL
LIN {X 0,Y 545.558,Z 424.248,A -85,B 0,C 180,E1 25715.126,E2 25715.126} C_VEL
LIN {X 0,Y 545.507,Z 424.255,A -85,B 0,C 180,E1 25711.896,E2 25711.896} C_VEL
LIN {X 0,Y 545.504,Z 424.273,A -85,B 0,C 180,E1 25708.466,E2 25708.466} C_VEL
LIN {X 0,Y 545.555,Z 424.275,A -85,B 0,C 180,E1 25705.195,E2 25705.195} C_VEL
LIN {X 0,Y 545.486,Z 424.274,A -85,B 0,C 180,E1 25701.983,E2 25701.983} C_VEL
LIN {X 0,Y 545.532,Z 424.193,A -85,B 0,C 180,E1 25698.852,E2 25698.852} C_VEL
LIN {X 0,Y 545.491,Z 424.323,A -85,B 0,C 180,E1 25695.645,E2 25695.645} C_VEL
LIN {X 0,Y 545.835,Z 425.753,A -85,B 0,C 180,E1 25695.407,E2 25695.407} C_VEL
LIN {X 0,Y 547.738,Z 428.858,A -85,B 0,C 180,E1 25695.126,E2 25695.126} C_VEL
LIN {X 0,Y 549.379,Z 430.582,A -85,B 0,C 180,E1 25694.909,E2 25694.909} C_VEL
LIN {X 0,Y 552.038,Z 434.522,A -85,B 0,C 180,E1 25694.542,E2 25694.542} C_VEL
LIN {X 0,Y 554.111,Z 437.425,A -85,B 0,C 180,E1 25694.261,E2 25694.261} C_VEL
LIN {X 0,Y 560.265,Z 445.756,A -85,B 0,C 180,E1 25693.455,E2 25693.455} C_VEL
LIN {X 0,Y 573.329,Z 464.814,A -85,B 0,C 180,E1 25691.811,E2 25691.811} C_VEL
LIN {X 0,Y 583.659,Z 481.045,A -85,B 0,C 180,E1 25690.574,E2 25690.574} C_VEL
LIN {X 0,Y 587.085,Z 487.269,A -85,B 0,C 180,E1 25690.165,E2 25690.165} C_VEL
LIN {X 0,Y 580.649,Z 736.438,A -85,B 0,C 180,E1 25686.75,E2 25686.75} C_VEL
LIN {X 0,Y 580.203,Z 753.992,A -85,B 0,C 180,E1 25686.512,E2 25686.512} C_VEL
LIN {X 0,Y 579.231,Z 761.687,A -85,B 0,C 180,E1 25686.469,E2 25686.469} C_VEL
LIN {X 0,Y 573.813,Z 782.208,A -85,B 0,C 180,E1 25686.581,E2 25686.581} C_VEL
LIN {X 0,Y 573.077,Z 788.809,A -85,B 0,C 180,E1 25686.536,E2 25686.536} C_VEL
LIN {X 0,Y 571.981,Z 817.649,A -85,B 0,C 180,E1 25686.071,E2 25686.071} C_VEL
LIN {X 0,Y 570.719,Z 837.944,A -85,B 0,C 180,E1 25685.614,E2 25685.614} C_VEL
LIN {X 0,Y 568.872,Z 861.427,A -85,B 0,C 180,E1 25684.929,E2 25684.929} C_VEL
LIN {X 0,Y 566.753,Z 882.9,A -85,B 0,C 180,E1 25684.127,E2 25684.127} C_VEL
LIN {X 0,Y 564.504,Z 902.786,A -85,B 0,C 180,E1 25683.244,E2 25683.244} C_VEL
LIN {X 0,Y 561.504,Z 926.288,A -85,B 0,C 180,E1 25681.99,E2 25681.99} C_VEL
LIN {X 0,Y 558.807,Z 945.506,A -85,B 0,C 180,E1 25680.781,E2 25680.781} C_VEL
LIN {X 0,Y 555.467,Z 967.788,A -85,B 0,C 180,E1 25679.139,E2 25679.139} C_VEL
LIN {X 0,Y 552.792,Z 984.646,A -85,B 0,C 180,E1 25677.701,E2 25677.701} C_VEL
LIN {X 0,Y 549.67,Z 1003.851,A -85,B 0,C 180,E1 25675.828,E2 25675.828} C_VEL
LIN {X 0,Y 547.096,Z 1019.587,A -85,B 0,C 180,E1 25674.052,E2 25674.052} C_VEL
LIN {X 0,Y 544.524,Z 1035.779,A -85,B 0,C 180,E1 25671.979,E2 25671.979} C_VEL
LIN {X 0,Y 542.288,Z 1050.158,A -85,B 0,C 180,E1 25669.832,E2 25669.832} C_VEL
LIN {X 0,Y 540.376,Z 1063.543,A -85,B 0,C 180,E1 25667.554,E2 25667.554} C_VEL
LIN {X 0,Y 538.828,Z 1075.371,A -85,B 0,C 180,E1 25665.168,E2 25665.168} C_VEL
LIN {X 0,Y 537.71,Z 1085.57,A -85,B 0,C 180,E1 25662.785,E2 25662.785} C_VEL
LIN {X 0,Y 536.887,Z 1094.324,A -85,B 0,C 180,E1 25660.299,E2 25660.299} C_VEL
LIN {X 0,Y 536.424,Z 1100.957,A -85,B 0,C 180,E1 25658.036,E2 25658.036} C_VEL
LIN {X 0,Y 536.103,Z 1107.142,A -85,B 0,C 180,E1 25655.351,E2 25655.351} C_VEL
LIN {X 0,Y 535.971,Z 1110.953,A -85,B 0,C 180,E1 25653.101,E2 25653.101} C_VEL
LIN {X 0,Y 535.921,Z 1113.73,A -85,B 0,C 180,E1 25650.748,E2 25650.748} C_VEL
LIN {X 0,Y 535.921,Z 1115.215,A -85,B 0,C 180,E1 25648.075,E2 25648.075} C_VEL
LIN {X 0,Y 535.919,Z 1115.216,A -85,B 0,C 180,E1 25645.827,E2 25645.827} C_VEL
LIN {X 0,Y 535.919,Z 1113.718,A -85,B 0,C 180,E1 25643.142,E2 25643.142} C_VEL
LIN {X 0,Y 535.974,Z 1111.064,A -85,B 0,C 180,E1 25640.876,E2 25640.876} C_VEL
LIN {X 0,Y 536.102,Z 1107.23,A -85,B 0,C 180,E1 25638.597,E2 25638.597} C_VEL
LIN {X 0,Y 536.424,Z 1100.962,A -85,B 0,C 180,E1 25635.866,E2 25635.866} C_VEL
LIN {X 0,Y 536.875,Z 1094.534,A -85,B 0,C 180,E1 25633.666,E2 25633.666} C_VEL
LIN {X 0,Y 537.691,Z 1085.835,A -85,B 0,C 180,E1 25631.181,E2 25631.181} C_VEL
LIN {X 0,Y 538.809,Z 1075.613,A -85,B 0,C 180,E1 25628.785,E2 25628.785} C_VEL
LIN {X 0,Y 540.324,Z 1064.06,A -85,B 0,C 180,E1 25626.439,E2 25626.439} C_VEL
LIN {X 0,Y 542.308,Z 1050.395,A -85,B 0,C 180,E1 25624.089,E2 25624.089} C_VEL
LIN {X 0,Y 544.541,Z 1036.268,A -85,B 0,C 180,E1 25621.961,E2 25621.961} C_VEL
LIN {X 0,Y 547.217,Z 1019.852,A -85,B 0,C 180,E1 25619.835,E2 25619.835} C_VEL
LIN {X 0,Y 549.944,Z 1003.684,A -85,B 0,C 180,E1 25617.995,E2 25617.995} C_VEL
LIN {X 0,Y 553.072,Z 985.071,A -85,B 0,C 180,E1 25616.163,E2 25616.163} C_VEL
LIN {X 0,Y 555.918,Z 967.752,A -85,B 0,C 180,E1 25614.672,E2 25614.672} C_VEL
LIN {X 0,Y 559.341,Z 945.822,A -85,B 0,C 180,E1 25613.042,E2 25613.042} C_VEL
LIN {X 0,Y 562.104,Z 926.875,A -85,B 0,C 180,E1 25611.836,E2 25611.836} C_VEL
LIN {X 0,Y 565.232,Z 903.544,A -85,B 0,C 180,E1 25610.575,E2 25610.575} C_VEL
LIN {X 0,Y 567.649,Z 883.119,A -85,B 0,C 180,E1 25609.659,E2 25609.659} C_VEL
LIN {X 0,Y 569.979,Z 860.612,A -85,B 0,C 180,E1 25608.814,E2 25608.814} C_VEL
LIN {X 0,Y 571.855,Z 837.409,A -85,B 0,C 180,E1 25608.141,E2 25608.141} C_VEL
LIN {X 0,Y 573.199,Z 816.669,A -85,B 0,C 180,E1 25607.674,E2 25607.674} C_VEL
LIN {X 0,Y 574.415,Z 784.394,A -85,B 0,C 180,E1 25607.165,E2 25607.165} C_VEL
LIN {X 0,Y 581.575,Z 537.146,A -85,B 0,C 180,E1 25603.714,E2 25603.714} C_VEL
LIN {X 0,Y 582.863,Z 490.487,A -85,B 0,C 180,E1 25603.043,E2 25603.043} C_VEL
LIN {X 0,Y 573.15,Z 474.92,A -85,B 0,C 180,E1 25601.775,E2 25601.775} C_VEL
LIN {X 0,Y 560.242,Z 456.476,A -85,B 0,C 180,E1 25600.013,E2 25600.013} C_VEL
LIN {X 0,Y 552.374,Z 445.981,A -85,B 0,C 180,E1 25598.879,E2 25598.879} C_VEL
LIN {X 0,Y 548.664,Z 441.01,A -85,B 0,C 180,E1 25598.322,E2 25598.322} C_VEL
LIN {X 0,Y 545.137,Z 436.315,A -85,B 0,C 180,E1 25597.78,E2 25597.78} C_VEL
